LIN {X 0,Y 418.329,Z 253.378,A -85,B 0,C 180,E1 -10089.672,E2 -10089.672} C_VEL
LIN {X 0,Y 418.34,Z 253.367,A -85,B 0,C 180,E1 -10093,E2 -10093} C_VEL
LIN {X 0,Y 418.305,Z 253.377,A -85,B 0,C 180,E1 -10096.734,E2 -10096.734} C_VEL
LIN {X 0,Y 418.264,Z 253.384,A -85,B 0,C 180,E1 -10099.79,E2 -10099.79} C_VEL
LIN {X 0,Y 418.221,Z 253.385,A -85,B 0,C 180,E1 -10102.737,E2 -10102.737} C_VEL
LIN {X 0,Y 418.211,Z 253.382,A -85,B 0,C 180,E1 -10105.908,E2 -10105.908} C_VEL
LIN {X 0,Y 418.25,Z 253.38,A -85,B 0,C 180,E1 -10109.163,E2 -10109.163} C_VEL
LIN {X 0,Y 418.243,Z 253.379,A -85,B 0,C 180,E1 -10112.842,E2 -10112.842} C_VEL
LIN {X 0,Y 418.234,Z 253.386,A -85,B 0,C 180,E1 -10116.237,E2 -10116.237} C_VEL
LIN {X 0,Y 418.194,Z 253.389,A -85,B 0,C 180,E1 -10119.688,E2 -10119.688} C_VEL
LIN {X 0,Y 418.203,Z 253.392,A -85,B 0,C 180,E1 -10122.318,E2 -10122.318} C_VEL
LIN {X 0,Y 418.231,Z 253.389,A -85,B 0,C 180,E1 -10125.109,E2 -10125.109} C_VEL
LIN {X 0,Y 418.214,Z 253.389,A -85,B 0,C 180,E1 -10127.764,E2 -10127.764} C_VEL
LIN {X 0,Y 418.228,Z 253.376,A -85,B 0,C 180,E1 -10131.556,E2 -10131.556} C_VEL
LIN {X 0,Y 418.247,Z 253.374,A -85,B 0,C 180,E1 -10135.158,E2 -10135.158} C_VEL
LIN {X 0,Y 418.237,Z 253.538,A -85,B 0,C 180,E1 -10138.483,E2 -10138.483} C_VEL
LIN {X 0,Y 421.565,Z 267.775,A -85,B 0,C 180,E1 -10141.088,E2 -10141.088} C_VEL
LIN {X 0,Y 422.679,Z 274.559,A -85,B 0,C 180,E1 -10142.254,E2 -10142.254} C_VEL
LIN {X 0,Y 421.513,Z 292.793,A -85,B 0,C 180,E1 -10145.102,E2 -10145.102} C_VEL
LIN {X 0,Y 420.246,Z 314.263,A -85,B 0,C 180,E1 -10148.413,E2 -10148.413} C_VEL
LIN {X 0,Y 419.602,Z 328.237,A -85,B 0,C 180,E1 -10150.523,E2 -10150.523} C_VEL
LIN {X 0,Y 423.082,Z 354.453,A -85,B 0,C 180,E1 -10151.189,E2 -10151.189} C_VEL
LIN {X 0,Y 424.096,Z 367.083,A -85,B 0,C 180,E1 -10151.465,E2 -10151.465} C_VEL
LIN {X 0,Y 423.18,Z 439.314,A -85,B 0,C 180,E1 -10152.731,E2 -10152.731} C_VEL
LIN {X 0,Y 422.504,Z 453.178,A -85,B 0,C 180,E1 -10153.17,E2 -10153.17} C_VEL
LIN {X 0,Y 421.636,Z 466.154,A -85,B 0,C 180,E1 -10153.788,E2 -10153.788} C_VEL
LIN {X 0,Y 420.772,Z 478.778,A -85,B 0,C 180,E1 -10154.624,E2 -10154.624} C_VEL
LIN {X 0,Y 419.851,Z 490.068,A -85,B 0,C 180,E1 -10155.582,E2 -10155.582} C_VEL
LIN {X 0,Y 419.119,Z 500.694,A -85,B 0,C 180,E1 -10156.719,E2 -10156.719} C_VEL
LIN {X 0,Y 418.384,Z 509.542,A -85,B 0,C 180,E1 -10157.879,E2 -10157.879} C_VEL
LIN {X 0,Y 417.84,Z 518.608,A -85,B 0,C 180,E1 -10159.338,E2 -10159.338} C_VEL
LIN {X 0,Y 417.516,Z 525.95,A -85,B 0,C 180,E1 -10160.798,E2 -10160.798} C_VEL
LIN {X 0,Y 417.368,Z 531.851,A -85,B 0,C 180,E1 -10162.258,E2 -10162.258} C_VEL
LIN {X 0,Y 417.325,Z 536.784,A -85,B 0,C 180,E1 -10163.812,E2 -10163.812} C_VEL
LIN {X 0,Y 417.357,Z 540.104,A -85,B 0,C 180,E1 -10165.17,E2 -10165.17} C_VEL
LIN {X 0,Y 417.497,Z 541.913,A -85,B 0,C 180,E1 -10166.139,E2 -10166.139} C_VEL
LIN {X 0,Y 417.534,Z 543.293,A -85,B 0,C 180,E1 -10167.105,E2 -10167.105} C_VEL
LIN {X 0,Y 417.524,Z 544.828,A -85,B 0,C 180,E1 -10169.035,E2 -10169.035} C_VEL
LIN {X 0,Y 417.577,Z 544.955,A -85,B 0,C 180,E1 -10170,E2 -10170} C_VEL
LIN {X 0,Y 417.543,Z 544.671,A -85,B 0,C 180,E1 -10170.964,E2 -10170.964} C_VEL
LIN {X 0,Y 417.521,Z 543.992,A -85,B 0,C 180,E1 -10171.929,E2 -10171.929} C_VEL
LIN {X 0,Y 417.552,Z 542.91,A -85,B 0,C 180,E1 -10172.894,E2 -10172.894} C_VEL
LIN {X 0,Y 417.509,Z 540.432,A -85,B 0,C 180,E1 -10174.344,E2 -10174.344} C_VEL
LIN {X 0,Y 417.444,Z 536.915,A -85,B 0,C 180,E1 -10175.797,E2 -10175.797} C_VEL
LIN {X 0,Y 417.412,Z 532.283,A -85,B 0,C 180,E1 -10177.254,E2 -10177.254} C_VEL
LIN {X 0,Y 417.487,Z 525.258,A -85,B 0,C 180,E1 -10178.958,E2 -10178.958} C_VEL
LIN {X 0,Y 417.764,Z 517.649,A -85,B 0,C 180,E1 -10180.418,E2 -10180.418} C_VEL
LIN {X 0,Y 418.142,Z 509.905,A -85,B 0,C 180,E1 -10181.635,E2 -10181.635} C_VEL
LIN {X 0,Y 418.73,Z 501.162,A -85,B 0,C 180,E1 -10182.774,E2 -10182.774} C_VEL
LIN {X 0,Y 419.276,Z 491.428,A -85,B 0,C 180,E1 -10183.819,E2 -10183.819} C_VEL
LIN {X 0,Y 419.967,Z 480.199,A -85,B 0,C 180,E1 -10184.785,E2 -10184.785} C_VEL
LIN {X 0,Y 420.71,Z 467.631,A -85,B 0,C 180,E1 -10185.626,E2 -10185.626} C_VEL
LIN {X 0,Y 421.417,Z 455.695,A -85,B 0,C 180,E1 -10186.22,E2 -10186.22} C_VEL
LIN {X 0,Y 421.986,Z 442.65,A -85,B 0,C 180,E1 -10186.664,E2 -10186.664} C_VEL
LIN {X 0,Y 422.225,Z 424.048,A -85,B 0,C 180,E1 -10187.028,E2 -10187.028} C_VEL
LIN {X 0,Y 422.691,Z 362.653,A -85,B 0,C 180,E1 -10188.064,E2 -10188.064} C_VEL
LIN {X 0,Y 419.121,Z 329.102,A -85,B 0,C 180,E1 -10188.799,E2 -10188.799} C_VEL
LIN {X 0,Y 419.927,Z 308.584,A -85,B 0,C 180,E1 -10191.862,E2 -10191.862} C_VEL
LIN {X 0,Y 421.052,Z 286.579,A -85,B 0,C 180,E1 -10195.19,E2 -10195.19} C_VEL
LIN {X 0,Y 421.815,Z 271.199,A -85,B 0,C 180,E1 -10197.538,E2 -10197.538} C_VEL
LIN {X 0,Y 418.56,Z 254.958,A -85,B 0,C 180,E1 -10200.246,E2 -10200.246} C_VEL
LIN {X 0,Y 418.271,Z 253.461,A -85,B 0,C 180,E1 -10200.571,E2 -10200.571} C_VEL
LIN {X 0,Y 418.226,Z 253.391,A -85,B 0,C 180,E1 -10203.678,E2 -10203.678} C_VEL
LIN {X 0,Y 418.225,Z 253.39,A -85,B 0,C 180,E1 -10207.224,E2 -10207.224} C_VEL
LIN {X 0,Y 418.199,Z 253.391,A -85,B 0,C 180,E1 -10210.949,E2 -10210.949} C_VEL
LIN {X 0,Y 418.193,Z 253.391,A -85,B 0,C 180,E1 -10213.727,E2 -10213.727} C_VEL
LIN {X 0,Y 418.19,Z 253.39,A -85,B 0,C 180,E1 -10216.446,E2 -10216.446} C_VEL
LIN {X 0,Y 418.198,Z 253.395,A -85,B 0,C 180,E1 -10219.132,E2 -10219.132} C_VEL
LIN {X 0,Y 418.224,Z 253.388,A -85,B 0,C 180,E1 -10222.774,E2 -10222.774} C_VEL
LIN {X 0,Y 418.217,Z 253.386,A -85,B 0,C 180,E1 -10226.32,E2 -10226.32} C_VEL
LIN {X 0,Y 418.226,Z 253.385,A -85,B 0,C 180,E1 -10229.726,E2 -10229.726} C_VEL
LIN {X 0,Y 418.19,Z 253.396,A -85,B 0,C 180,E1 -10233.015,E2 -10233.015} C_VEL
LIN {X 0,Y 418.243,Z 253.383,A -85,B 0,C 180,E1 -10236.216,E2 -10236.216} C_VEL
LIN {X 0,Y 418.235,Z 253.386,A -85,B 0,C 180,E1 -10239.336,E2 -10239.336} C_VEL
LIN {X 0,Y 418.265,Z 253.383,A -85,B 0,C 180,E1 -10242.395,E2 -10242.395} C_VEL
LIN {X 0,Y 418.28,Z 253.379,A -85,B 0,C 180,E1 -10245.402,E2 -10245.402} C_VEL
LIN {X 0,Y 418.298,Z 253.379,A -85,B 0,C 180,E1 -10248.369,E2 -10248.369} C_VEL
LIN {X 0,Y 418.434,Z 253.362,A -85,B 0,C 180,E1 -10252.278,E2 -10252.278} C_VEL
LIN {X 0,Y 418.45,Z 253.36,A -85,B 0,C 180,E1 -10254.217,E2 -10254.217} C_VEL
LIN {X 0,Y 418.523,Z 253.35,A -85,B 0,C 180,E1 -10258.076,E2 -10258.076} C_VEL
LIN {X 0,Y 418.458,Z 253.358,A -85,B 0,C 180,E1 -10260.963,E2 -10260.963} C_VEL
LIN {X 0,Y 418.453,Z 253.359,A -85,B 0,C 180,E1 -10262.888,E2 -10262.888} C_VEL
LIN {X 0,Y 418.424,Z 253.362,A -85,B 0,C 180,E1 -10266.617,E2 -10266.617} C_VEL
LIN {X 0,Y 418.306,Z 253.376,A -85,B 0,C 180,E1 -10269.672,E2 -10269.672} C_VEL
LIN {X 0,Y 418.334,Z 253.372,A -85,B 0,C 180,E1 -10273,E2 -10273} C_VEL
LIN {X 0,Y 418.3,Z 253.377,A -85,B 0,C 180,E1 -10276.735,E2 -10276.735} C_VEL
LIN {X 0,Y 418.259,Z 253.383,A -85,B 0,C 180,E1 -10279.79,E2 -10279.79} C_VEL
LIN {X 0,Y 418.217,Z 253.387,A -85,B 0,C 180,E1 -10282.738,E2 -10282.738} C_VEL
LIN {X 0,Y 418.207,Z 253.392,A -85,B 0,C 180,E1 -10285.909,E2 -10285.909} C_VEL
LIN {X 0,Y 418.247,Z 253.382,A -85,B 0,C 180,E1 -10289.164,E2 -10289.164} C_VEL
LIN {X 0,Y 418.231,Z 253.386,A -85,B 0,C 180,E1 -10292.53,E2 -10292.53} C_VEL
LIN {X 0,Y 418.241,Z 253.383,A -85,B 0,C 180,E1 -10294.843,E2 -10294.843} C_VEL
LIN {X 0,Y 418.224,Z 253.386,A -85,B 0,C 180,E1 -10298.446,E2 -10298.446} C_VEL
LIN {X 0,Y 418.21,Z 253.389,A -85,B 0,C 180,E1 -10302.237,E2 -10302.237} C_VEL
LIN {X 0,Y 418.228,Z 253.385,A -85,B 0,C 180,E1 -10305.11,E2 -10305.11} C_VEL
LIN {X 0,Y 418.212,Z 253.394,A -85,B 0,C 180,E1 -10307.765,E2 -10307.765} C_VEL
LIN {X 0,Y 418.228,Z 253.391,A -85,B 0,C 180,E1 -10311.557,E2 -10311.557} C_VEL
LIN {X 0,Y 418.244,Z 253.385,A -85,B 0,C 180,E1 -10315.159,E2 -10315.159} C_VEL
LIN {X 0,Y 418.229,Z 253.391,A -85,B 0,C 180,E1 -10317.472,E2 -10317.472} C_VEL
LIN {X 0,Y 418.256,Z 253.382,A -85,B 0,C 180,E1 -10320.9,E2 -10320.9} C_VEL
LIN {X 0,Y 418.209,Z 253.388,A -85,B 0,C 180,E1 -10324.093,E2 -10324.093} C_VEL
LIN {X 0,Y 418.232,Z 253.389,A -85,B 0,C 180,E1 -10327.553,E2 -10327.553} C_VEL
LIN {X 0,Y 418.252,Z 253.382,A -85,B 0,C 180,E1 -10330.364,E2 -10330.364} C_VEL
LIN {X 0,Y 418.281,Z 253.384,A -85,B 0,C 180,E1 -10333.404,E2 -10333.404} C_VEL
LIN {X 0,Y 418.349,Z 253.377,A -85,B 0,C 180,E1 -10337.386,E2 -10337.386} C_VEL
LIN {X 0,Y 418.353,Z 253.613,A -85,B 0,C 180,E1 -10339.517,E2 -10339.517} C_VEL
LIN {X 0,Y 418.633,Z 254.814,A -85,B 0,C 180,E1 -10339.664,E2 -10339.664} C_VEL
LIN {X 0,Y 423.488,Z 268.312,A -85,B 0,C 180,E1 -10340.107,E2 -10340.107} C_VEL
LIN {X 0,Y 422.736,Z 341.816,A -85,B 0,C 180,E1 -10341.375,E2 -10341.375} C_VEL
LIN {X 0,Y 422.651,Z 355.208,A -85,B 0,C 180,E1 -10341.815,E2 -10341.815} C_VEL
LIN {X 0,Y 422.338,Z 366.469,A -85,B 0,C 180,E1 -10342.35,E2 -10342.35} C_VEL
LIN {X 0,Y 421.96,Z 377.78,A -85,B 0,C 180,E1 -10343.065,E2 -10343.065} C_VEL
LIN {X 0,Y 421.365,Z 389.414,A -85,B 0,C 180,E1 -10344.017,E2 -10344.017} C_VEL
LIN {X 0,Y 420.76,Z 399.809,A -85,B 0,C 180,E1 -10345.09,E2 -10345.09} C_VEL
LIN {X 0,Y 420.249,Z 408.305,A -85,B 0,C 180,E1 -10346.165,E2 -10346.165} C_VEL
LIN {X 0,Y 419.828,Z 414.206,A -85,B 0,C 180,E1 -10347.043,E2 -10347.043} C_VEL
LIN {X 0,Y 418.927,Z 418,A -85,B 0,C 180,E1 -10347.654,E2 -10347.654} C_VEL
LIN {X 0,Y 415.715,Z 423.87,A -85,B 0,C 180,E1 -10348.66,E2 -10348.66} C_VEL
LIN {X 0,Y 412.503,Z 429.122,A -85,B 0,C 180,E1 -10349.735,E2 -10349.735} C_VEL
LIN {X 0,Y 411.616,Z 431.916,A -85,B 0,C 180,E1 -10350.444,E2 -10350.444} C_VEL
LIN {X 0,Y 411.325,Z 436.709,A -85,B 0,C 180,E1 -10351.959,E2 -10351.959} C_VEL
LIN {X 0,Y 411.028,Z 440.273,A -85,B 0,C 180,E1 -10353.431,E2 -10353.431} C_VEL
LIN {X 0,Y 411.014,Z 442.819,A -85,B 0,C 180,E1 -10354.905,E2 -10354.905} C_VEL
LIN {X 0,Y 410.93,Z 444.038,A -85,B 0,C 180,E1 -10355.89,E2 -10355.89} C_VEL
LIN {X 0,Y 410.866,Z 444.998,A -85,B 0,C 180,E1 -10357.198,E2 -10357.198} C_VEL
LIN {X 0,Y 410.864,Z 445.251,A -85,B 0,C 180,E1 -10358.856,E2 -10358.856} C_VEL
LIN {X 0,Y 410.918,Z 444.89,A -85,B 0,C 180,E1 -10359.848,E2 -10359.848} C_VEL
LIN {X 0,Y 410.983,Z 444.108,A -85,B 0,C 180,E1 -10360.842,E2 -10360.842} C_VEL
LIN {X 0,Y 411.326,Z 441.302,A -85,B 0,C 180,E1 -10362.834,E2 -10362.834} C_VEL
LIN {X 0,Y 411.645,Z 438.051,A -85,B 0,C 180,E1 -10364.333,E2 -10364.333} C_VEL
LIN {X 0,Y 412.072,Z 433.706,A -85,B 0,C 180,E1 -10365.836,E2 -10365.836} C_VEL
LIN {X 0,Y 412.7,Z 427.4,A -85,B 0,C 180,E1 -10367.512,E2 -10367.512} C_VEL
LIN {X 0,Y 413.481,Z 419.712,A -85,B 0,C 180,E1 -10369.099,E2 -10369.099} C_VEL
LIN {X 0,Y 414.137,Z 412.184,A -85,B 0,C 180,E1 -10370.358,E2 -10370.358} C_VEL
LIN {X 0,Y 414.964,Z 402.642,A -85,B 0,C 180,E1 -10371.659,E2 -10371.659} C_VEL
LIN {X 0,Y 415.666,Z 392.66,A -85,B 0,C 180,E1 -10372.753,E2 -10372.753} C_VEL
LIN {X 0,Y 416.294,Z 382.696,A -85,B 0,C 180,E1 -10373.638,E2 -10373.638} C_VEL
LIN {X 0,Y 416.958,Z 370.814,A -85,B 0,C 180,E1 -10374.467,E2 -10374.467} C_VEL
LIN {X 0,Y 417.371,Z 358.128,A -85,B 0,C 180,E1 -10375.128,E2 -10375.128} C_VEL
LIN {X 0,Y 417.56,Z 345.349,A -85,B 0,C 180,E1 -10375.583,E2 -10375.583} C_VEL
LIN {X 0,Y 417.672,Z 324.353,A -85,B 0,C 180,E1 -10376.004,E2 -10376.004} C_VEL
LIN {X 0,Y 418.487,Z 271.987,A -85,B 0,C 180,E1 -10376.91,E2 -10376.91} C_VEL
LIN {X 0,Y 411.384,Z 255.243,A -85,B 0,C 180,E1 -10377.651,E2 -10377.651} C_VEL
LIN {X 0,Y 411.205,Z 254.336,A -85,B 0,C 180,E1 -10377.862,E2 -10377.862} C_VEL
LIN {X 0,Y 411.19,Z 254.242,A -85,B 0,C 180,E1 -10380.847,E2 -10380.847} C_VEL
LIN {X 0,Y 411.194,Z 254.26,A -85,B 0,C 180,E1 -10384.334,E2 -10384.334} C_VEL
LIN {X 0,Y 411.188,Z 254.232,A -85,B 0,C 180,E1 -10386.742,E2 -10386.742} C_VEL
LIN {X 0,Y 411.168,Z 254.268,A -85,B 0,C 180,E1 -10389.719,E2 -10389.719} C_VEL
LIN {X 0,Y 411.162,Z 254.269,A -85,B 0,C 180,E1 -10393.134,E2 -10393.134} C_VEL
LIN {X 0,Y 411.162,Z 254.263,A -85,B 0,C 180,E1 -10395.881,E2 -10395.881} C_VEL
LIN {X 0,Y 411.146,Z 254.273,A -85,B 0,C 180,E1 -10398.774,E2 -10398.774} C_VEL
LIN {X 0,Y 411.179,Z 254.251,A -85,B 0,C 180,E1 -10402.024,E2 -10402.024} C_VEL
LIN {X 0,Y 411.202,Z 254.263,A -85,B 0,C 180,E1 -10405.666,E2 -10405.666} C_VEL
LIN {X 0,Y 411.185,Z 254.243,A -85,B 0,C 180,E1 -10409.152,E2 -10409.152} C_VEL
LIN {X 0,Y 411.172,Z 254.257,A -85,B 0,C 180,E1 -10411.406,E2 -10411.406} C_VEL
LIN {X 0,Y 411.212,Z 254.258,A -85,B 0,C 180,E1 -10414.932,E2 -10414.932} C_VEL
LIN {X 0,Y 411.199,Z 254.235,A -85,B 0,C 180,E1 -10417.913,E2 -10417.913} C_VEL
LIN {X 0,Y 411.217,Z 254.254,A -85,B 0,C 180,E1 -10421.051,E2 -10421.051} C_VEL
LIN {X 0,Y 411.247,Z 254.255,A -85,B 0,C 180,E1 -10424.131,E2 -10424.131} C_VEL
LIN {X 0,Y 411.297,Z 254.248,A -85,B 0,C 180,E1 -10427.165,E2 -10427.165} C_VEL
LIN {X 0,Y 411.281,Z 254.245,A -85,B 0,C 180,E1 -10430.161,E2 -10430.161} C_VEL
LIN {X 0,Y 411.383,Z 254.239,A -85,B 0,C 180,E1 -10433.131,E2 -10433.131} C_VEL
LIN {X 0,Y 411.278,Z 254.25,A -85,B 0,C 180,E1 -10435.098,E2 -10435.098} C_VEL
LIN {X 0,Y 411.494,Z 254.228,A -85,B 0,C 180,E1 -10438.042,E2 -10438.042} C_VEL
LIN {X 0,Y 411.369,Z 254.237,A -85,B 0,C 180,E1 -10440.979,E2 -10440.979} C_VEL
LIN {X 0,Y 411.431,Z 254.227,A -85,B 0,C 180,E1 -10442.937,E2 -10442.937} C_VEL
LIN {X 0,Y 411.378,Z 254.235,A -85,B 0,C 180,E1 -10446.868,E2 -10446.868} C_VEL
LIN {X 0,Y 411.281,Z 254.254,A -85,B 0,C 180,E1 -10449.839,E2 -10449.839} C_VEL
LIN {X 0,Y 411.299,Z 254.244,A -85,B 0,C 180,E1 -10453.104,E2 -10453.104} C_VEL
LIN {X 0,Y 411.252,Z 254.257,A -85,B 0,C 180,E1 -10456.889,E2 -10456.889} C_VEL
LIN {X 0,Y 411.225,Z 254.259,A -85,B 0,C 180,E1 -10459.987,E2 -10459.987} C_VEL
LIN {X 0,Y 411.181,Z 254.266,A -85,B 0,C 180,E1 -10463.149,E2 -10463.149} C_VEL
LIN {X 0,Y 411.165,Z 254.26,A -85,B 0,C 180,E1 -10466.386,E2 -10466.386} C_VEL
LIN {X 0,Y 411.189,Z 254.264,A -85,B 0,C 180,E1 -10469.714,E2 -10469.714} C_VEL
LIN {X 0,Y 411.199,Z 254.253,A -85,B 0,C 180,E1 -10473.156,E2 -10473.156} C_VEL
LIN {X 0,Y 411.184,Z 254.267,A -85,B 0,C 180,E1 -10476.552,E2 -10476.552} C_VEL
LIN {X 0,Y 411.163,Z 254.265,A -85,B 0,C 180,E1 -10479.72,E2 -10479.72} C_VEL
LIN {X 0,Y 411.158,Z 254.264,A -85,B 0,C 180,E1 -10483.136,E2 -10483.136} C_VEL
LIN {X 0,Y 411.159,Z 254.266,A -85,B 0,C 180,E1 -10485.882,E2 -10485.882} C_VEL
LIN {X 0,Y 411.154,Z 254.262,A -85,B 0,C 180,E1 -10489.493,E2 -10489.493} C_VEL
LIN {X 0,Y 411.176,Z 254.261,A -85,B 0,C 180,E1 -10492.025,E2 -10492.025} C_VEL
LIN {X 0,Y 411.199,Z 254.252,A -85,B 0,C 180,E1 -10495.124,E2 -10495.124} C_VEL
LIN {X 0,Y 411.228,Z 254.442,A -85,B 0,C 180,E1 -10498.148,E2 -10498.148} C_VEL
LIN {X 0,Y 414.174,Z 267.128,A -85,B 0,C 180,E1 -10500.522,E2 -10500.522} C_VEL
LIN {X 0,Y 415.815,Z 275.627,A -85,B 0,C 180,E1 -10502.029,E2 -10502.029} C_VEL
LIN {X 0,Y 414.635,Z 293.851,A -85,B 0,C 180,E1 -10504.929,E2 -10504.929} C_VEL
LIN {X 0,Y 413.205,Z 316.945,A -85,B 0,C 180,E1 -10508.55,E2 -10508.55} C_VEL
LIN {X 0,Y 412.71,Z 327.289,A -85,B 0,C 180,E1 -10510.132,E2 -10510.132} C_VEL
LIN {X 0,Y 416.221,Z 353.382,A -85,B 0,C 180,E1 -10510.821,E2 -10510.821} C_VEL
LIN {X 0,Y 417.433,Z 366.101,A -85,B 0,C 180,E1 -10511.114,E2 -10511.114} C_VEL
LIN {X 0,Y 416.44,Z 438.793,A -85,B 0,C 180,E1 -10512.411,E2 -10512.411} C_VEL
LIN {X 0,Y 415.764,Z 452.537,A -85,B 0,C 180,E1 -10512.857,E2 -10512.857} C_VEL
LIN {X 0,Y 414.898,Z 464.922,A -85,B 0,C 180,E1 -10513.454,E2 -10513.454} C_VEL
LIN {X 0,Y 414.034,Z 476.832,A -85,B 0,C 180,E1 -10514.241,E2 -10514.241} C_VEL
LIN {X 0,Y 413.079,Z 488.314,A -85,B 0,C 180,E1 -10515.214,E2 -10515.214} C_VEL
LIN {X 0,Y 412.292,Z 497.634,A -85,B 0,C 180,E1 -10516.193,E2 -10516.193} C_VEL
LIN {X 0,Y 411.597,Z 507.261,A -85,B 0,C 180,E1 -10517.426,E2 -10517.426} C_VEL
LIN {X 0,Y 410.939,Z 516.573,A -85,B 0,C 180,E1 -10518.907,E2 -10518.907} C_VEL
LIN {X 0,Y 410.492,Z 524.111,A -85,B 0,C 180,E1 -10520.391,E2 -10520.391} C_VEL
LIN {X 0,Y 410.29,Z 531.109,A -85,B 0,C 180,E1 -10522.123,E2 -10522.123} C_VEL
LIN {X 0,Y 410.314,Z 535.287,A -85,B 0,C 180,E1 -10523.437,E2 -10523.437} C_VEL
LIN {X 0,Y 410.279,Z 539.315,A -85,B 0,C 180,E1 -10525.086,E2 -10525.086} C_VEL
LIN {X 0,Y 410.427,Z 541.11,A -85,B 0,C 180,E1 -10526.072,E2 -10526.072} C_VEL
LIN {X 0,Y 410.483,Z 542.481,A -85,B 0,C 180,E1 -10527.055,E2 -10527.055} C_VEL
LIN {X 0,Y 410.436,Z 543.437,A -85,B 0,C 180,E1 -10528.037,E2 -10528.037} C_VEL
LIN {X 0,Y 410.471,Z 543.986,A -85,B 0,C 180,E1 -10529.019,E2 -10529.019} C_VEL
LIN {X 0,Y 410.528,Z 544.099,A -85,B 0,C 180,E1 -10530,E2 -10530} C_VEL
LIN {X 0,Y 410.492,Z 543.805,A -85,B 0,C 180,E1 -10530.981,E2 -10530.981} C_VEL
LIN {X 0,Y 410.47,Z 543.114,A -85,B 0,C 180,E1 -10531.962,E2 -10531.962} C_VEL
LIN {X 0,Y 410.503,Z 542.012,A -85,B 0,C 180,E1 -10532.944,E2 -10532.944} C_VEL
LIN {X 0,Y 410.443,Z 539.513,A -85,B 0,C 180,E1 -10534.419,E2 -10534.419} C_VEL
LIN {X 0,Y 410.378,Z 534.748,A -85,B 0,C 180,E1 -10536.316,E2 -10536.316} C_VEL
LIN {X 0,Y 410.333,Z 529.453,A -85,B 0,C 180,E1 -10537.875,E2 -10537.875} C_VEL
LIN {X 0,Y 410.494,Z 523.089,A -85,B 0,C 180,E1 -10539.36,E2 -10539.36} C_VEL
LIN {X 0,Y 410.813,Z 515.154,A -85,B 0,C 180,E1 -10540.846,E2 -10540.846} C_VEL
LIN {X 0,Y 411.373,Z 505.235,A -85,B 0,C 180,E1 -10542.33,E2 -10542.33} C_VEL
LIN {X 0,Y 411.908,Z 495.947,A -85,B 0,C 180,E1 -10543.458,E2 -10543.458} C_VEL
LIN {X 0,Y 412.624,Z 484.831,A -85,B 0,C 180,E1 -10544.549,E2 -10544.549} C_VEL
LIN {X 0,Y 413.411,Z 473.825,A -85,B 0,C 180,E1 -10545.403,E2 -10545.403} C_VEL
LIN {X 0,Y 414.149,Z 461.68,A -85,B 0,C 180,E1 -10546.133,E2 -10546.133} C_VEL
LIN {X 0,Y 414.796,Z 449.272,A -85,B 0,C 180,E1 -10546.676,E2 -10546.676} C_VEL
LIN {X 0,Y 415.238,Z 436.492,A -85,B 0,C 180,E1 -10547.038,E2 -10547.038} C_VEL
LIN {X 0,Y 415.864,Z 363.556,A -85,B 0,C 180,E1 -10548.301,E2 -10548.301} C_VEL
LIN {X 0,Y 412.124,Z 328.112,A -85,B 0,C 180,E1 -10549.098,E2 -10549.098} C_VEL
LIN {X 0,Y 413,Z 307.432,A -85,B 0,C 180,E1 -10552.248,E2 -10552.248} C_VEL
LIN {X 0,Y 414.179,Z 285.781,A -85,B 0,C 180,E1 -10555.579,E2 -10555.579} C_VEL
LIN {X 0,Y 414.84,Z 273.589,A -85,B 0,C 180,E1 -10557.469,E2 -10557.469} C_VEL
LIN {X 0,Y 413.688,Z 266.297,A -85,B 0,C 180,E1 -10558.68,E2 -10558.68} C_VEL
LIN {X 0,Y 411.244,Z 254.369,A -85,B 0,C 180,E1 -10560.77,E2 -10560.77} C_VEL
LIN {X 0,Y 411.186,Z 254.266,A -85,B 0,C 180,E1 -10564.334,E2 -10564.334} C_VEL
LIN {X 0,Y 411.179,Z 254.264,A -85,B 0,C 180,E1 -10566.742,E2 -10566.742} C_VEL
LIN {X 0,Y 411.156,Z 254.268,A -85,B 0,C 180,E1 -10569.718,E2 -10569.718} C_VEL
LIN {X 0,Y 411.153,Z 254.271,A -85,B 0,C 180,E1 -10573.134,E2 -10573.134} C_VEL
LIN {X 0,Y 411.155,Z 254.267,A -85,B 0,C 180,E1 -10575.881,E2 -10575.881} C_VEL
LIN {X 0,Y 411.149,Z 254.27,A -85,B 0,C 180,E1 -10579.492,E2 -10579.492} C_VEL
LIN {X 0,Y 411.173,Z 254.264,A -85,B 0,C 180,E1 -10582.024,E2 -10582.024} C_VEL
LIN {X 0,Y 411.19,Z 254.268,A -85,B 0,C 180,E1 -10585.123,E2 -10585.123} C_VEL
LIN {X 0,Y 411.143,Z 254.267,A -85,B 0,C 180,E1 -10588.001,E2 -10588.001} C_VEL
LIN {X 0,Y 411.158,Z 254.268,A -85,B 0,C 180,E1 -10591.405,E2 -10591.405} C_VEL
LIN {X 0,Y 411.176,Z 254.27,A -85,B 0,C 180,E1 -10594.941,E2 -10594.941} C_VEL
LIN {X 0,Y 411.19,Z 254.261,A -85,B 0,C 180,E1 -10597.913,E2 -10597.913} C_VEL
LIN {X 0,Y 411.205,Z 254.264,A -85,B 0,C 180,E1 -10601.051,E2 -10601.051} C_VEL
LIN {X 0,Y 411.233,Z 254.257,A -85,B 0,C 180,E1 -10604.131,E2 -10604.131} C_VEL
LIN {X 0,Y 411.291,Z 254.251,A -85,B 0,C 180,E1 -10607.165,E2 -10607.165} C_VEL
LIN {X 0,Y 411.267,Z 254.253,A -85,B 0,C 180,E1 -10610.161,E2 -10610.161} C_VEL
LIN {X 0,Y 411.372,Z 254.24,A -85,B 0,C 180,E1 -10613.132,E2 -10613.132} C_VEL
LIN {X 0,Y 411.272,Z 254.253,A -85,B 0,C 180,E1 -10615.099,E2 -10615.099} C_VEL
LIN {X 0,Y 411.492,Z 254.226,A -85,B 0,C 180,E1 -10618.043,E2 -10618.043} C_VEL
LIN {X 0,Y 411.487,Z 254.226,A -85,B 0,C 180,E1 -10621.958,E2 -10621.958} C_VEL
LIN {X 0,Y 411.372,Z 254.239,A -85,B 0,C 180,E1 -10626.618,E2 -10626.618} C_VEL
LIN {X 0,Y 411.293,Z 254.25,A -85,B 0,C 180,E1 -10628.847,E2 -10628.847} C_VEL
LIN {X 0,Y 411.26,Z 254.255,A -85,B 0,C 180,E1 -10631.834,E2 -10631.834} C_VEL
LIN {X 0,Y 411.241,Z 254.256,A -85,B 0,C 180,E1 -10634.854,E2 -10634.854} C_VEL
LIN {X 0,Y 411.233,Z 254.26,A -85,B 0,C 180,E1 -10637.916,E2 -10637.916} C_VEL
LIN {X 0,Y 411.185,Z 254.262,A -85,B 0,C 180,E1 -10641.035,E2 -10641.035} C_VEL
LIN {X 0,Y 411.18,Z 254.268,A -85,B 0,C 180,E1 -10644.219,E2 -10644.219} C_VEL
LIN {X 0,Y 411.136,Z 254.269,A -85,B 0,C 180,E1 -10647.487,E2 -10647.487} C_VEL
LIN {X 0,Y 411.186,Z 254.265,A -85,B 0,C 180,E1 -10649.714,E2 -10649.714} C_VEL
LIN {X 0,Y 411.196,Z 254.261,A -85,B 0,C 180,E1 -10653.157,E2 -10653.157} C_VEL
LIN {X 0,Y 411.18,Z 254.263,A -85,B 0,C 180,E1 -10656.553,E2 -10656.553} C_VEL
LIN {X 0,Y 411.159,Z 254.271,A -85,B 0,C 180,E1 -10659.721,E2 -10659.721} C_VEL
LIN {X 0,Y 411.155,Z 254.266,A -85,B 0,C 180,E1 -10663.137,E2 -10663.137} C_VEL
LIN {X 0,Y 411.157,Z 254.271,A -85,B 0,C 180,E1 -10665.883,E2 -10665.883} C_VEL
LIN {X 0,Y 411.152,Z 254.271,A -85,B 0,C 180,E1 -10669.494,E2 -10669.494} C_VEL
LIN {X 0,Y 411.176,Z 254.266,A -85,B 0,C 180,E1 -10672.026,E2 -10672.026} C_VEL
LIN {X 0,Y 411.196,Z 254.263,A -85,B 0,C 180,E1 -10675.125,E2 -10675.125} C_VEL
LIN {X 0,Y 411.151,Z 254.268,A -85,B 0,C 180,E1 -10678.003,E2 -10678.003} C_VEL
LIN {X 0,Y 411.167,Z 254.27,A -85,B 0,C 180,E1 -10681.407,E2 -10681.407} C_VEL
LIN {X 0,Y 411.187,Z 254.264,A -85,B 0,C 180,E1 -10684.943,E2 -10684.943} C_VEL
LIN {X 0,Y 411.2,Z 254.262,A -85,B 0,C 180,E1 -10687.914,E2 -10687.914} C_VEL
LIN {X 0,Y 411.19,Z 254.265,A -85,B 0,C 180,E1 -10691.051,E2 -10691.051} C_VEL
LIN {X 0,Y 411.199,Z 254.26,A -85,B 0,C 180,E1 -10694.13,E2 -10694.13} C_VEL
LIN {X 0,Y 411.298,Z 254.252,A -85,B 0,C 180,E1 -10697.166,E2 -10697.166} C_VEL
LIN {X 0,Y 411.305,Z 254.438,A -85,B 0,C 180,E1 -10699.216,E2 -10699.216} C_VEL
LIN {X 0,Y 411.451,Z 255.25,A -85,B 0,C 180,E1 -10699.359,E2 -10699.359} C_VEL
LIN {X 0,Y 416.769,Z 270.131,A -85,B 0,C 180,E1 -10699.865,E2 -10699.865} C_VEL
LIN {X 0,Y 415.912,Z 341.892,A -85,B 0,C 180,E1 -10701.113,E2 -10701.113} C_VEL
LIN {X 0,Y 415.833,Z 354.716,A -85,B 0,C 180,E1 -10701.527,E2 -10701.527} C_VEL
LIN {X 0,Y 415.49,Z 366.877,A -85,B 0,C 180,E1 -10702.101,E2 -10702.101} C_VEL
LIN {X 0,Y 415.102,Z 378.281,A -85,B 0,C 180,E1 -10702.828,E2 -10702.828} C_VEL
LIN {X 0,Y 414.481,Z 390.009,A -85,B 0,C 180,E1 -10703.795,E2 -10703.795} C_VEL
LIN {X 0,Y 413.848,Z 400.449,A -85,B 0,C 180,E1 -10704.885,E2 -10704.885} C_VEL
LIN {X 0,Y 413.272,Z 409.85,A -85,B 0,C 180,E1 -10706.1,E2 -10706.1} C_VEL
LIN {X 0,Y 412.706,Z 417.574,A -85,B 0,C 180,E1 -10707.316,E2 -10707.316} C_VEL
LIN {X 0,Y 412.092,Z 425.134,A -85,B 0,C 180,E1 -10708.779,E2 -10708.779} C_VEL
LIN {X 0,Y 411.616,Z 431.916,A -85,B 0,C 180,E1 -10710.444,E2 -10710.444} C_VEL
LIN {X 0,Y 410.74,Z 434.523,A -85,B 0,C 180,E1 -10711.174,E2 -10711.174} C_VEL
LIN {X 0,Y 406.248,Z 439.724,A -85,B 0,C 180,E1 -10712.87,E2 -10712.87} C_VEL
LIN {X 0,Y 404.233,Z 442.061,A -85,B 0,C 180,E1 -10713.903,E2 -10713.903} C_VEL
LIN {X 0,Y 403.925,Z 442.96,A -85,B 0,C 180,E1 -10714.444,E2 -10714.444} C_VEL
LIN {X 0,Y 403.876,Z 444.991,A -85,B 0,C 180,E1 -10715.993,E2 -10715.993} C_VEL
LIN {X 0,Y 403.799,Z 446.102,A -85,B 0,C 180,E1 -10718.004,E2 -10718.004} C_VEL
LIN {X 0,Y 403.848,Z 446.086,A -85,B 0,C 180,E1 -10719.011,E2 -10719.011} C_VEL
LIN {X 0,Y 403.897,Z 445.686,A -85,B 0,C 180,E1 -10720.021,E2 -10720.021} C_VEL
LIN {X 0,Y 404.135,Z 443.617,A -85,B 0,C 180,E1 -10722.045,E2 -10722.045} C_VEL
LIN {X 0,Y 404.403,Z 441.54,A -85,B 0,C 180,E1 -10723.29,E2 -10723.29} C_VEL
LIN {X 0,Y 404.823,Z 437.301,A -85,B 0,C 180,E1 -10725.094,E2 -10725.094} C_VEL
LIN {X 0,Y 405.353,Z 432.476,A -85,B 0,C 180,E1 -10726.623,E2 -10726.623} C_VEL
LIN {X 0,Y 405.982,Z 426.348,A -85,B 0,C 180,E1 -10728.156,E2 -10728.156} C_VEL
LIN {X 0,Y 406.807,Z 418.626,A -85,B 0,C 180,E1 -10729.687,E2 -10729.687} C_VEL
LIN {X 0,Y 407.571,Z 410.658,A -85,B 0,C 180,E1 -10730.965,E2 -10730.965} C_VEL
LIN {X 0,Y 408.378,Z 400.862,A -85,B 0,C 180,E1 -10732.248,E2 -10732.248} C_VEL
LIN {X 0,Y 409.154,Z 391.185,A -85,B 0,C 180,E1 -10733.27,E2 -10733.27} C_VEL
LIN {X 0,Y 409.84,Z 380.682,A -85,B 0,C 180,E1 -10734.168,E2 -10734.168} C_VEL
LIN {X 0,Y 410.457,Z 368.828,A -85,B 0,C 180,E1 -10734.952,E2 -10734.952} C_VEL
LIN {X 0,Y 410.829,Z 356.149,A -85,B 0,C 180,E1 -10735.574,E2 -10735.574} C_VEL
LIN {X 0,Y 410.973,Z 343.681,A -85,B 0,C 180,E1 -10735.99,E2 -10735.99} C_VEL
LIN {X 0,Y 411.355,Z 306.087,A -85,B 0,C 180,E1 -10736.684,E2 -10736.684} C_VEL
LIN {X 0,Y 411.883,Z 273.341,A -85,B 0,C 180,E1 -10737.261,E2 -10737.261} C_VEL
LIN {X 0,Y 404.311,Z 256.008,A -85,B 0,C 180,E1 -10738.068,E2 -10738.068} C_VEL
LIN {X 0,Y 404.173,Z 255.199,A -85,B 0,C 180,E1 -10738.283,E2 -10738.283} C_VEL
LIN {X 0,Y 404.14,Z 255.12,A -85,B 0,C 180,E1 -10741.557,E2 -10741.557} C_VEL
LIN {X 0,Y 404.174,Z 255.12,A -85,B 0,C 180,E1 -10745.017,E2 -10745.017} C_VEL
LIN {X 0,Y 404.134,Z 255.136,A -85,B 0,C 180,E1 -10748.759,E2 -10748.759} C_VEL
LIN {X 0,Y 404.106,Z 255.139,A -85,B 0,C 180,E1 -10751.596,E2 -10751.596} C_VEL
LIN {X 0,Y 404.142,Z 255.147,A -85,B 0,C 180,E1 -10754.521,E2 -10754.521} C_VEL
LIN {X 0,Y 404.119,Z 255.134,A -85,B 0,C 180,E1 -10757.293,E2 -10757.293} C_VEL
LIN {X 0,Y 404.131,Z 255.145,A -85,B 0,C 180,E1 -10759.95,E2 -10759.95} C_VEL
LIN {X 0,Y 404.128,Z 255.13,A -85,B 0,C 180,E1 -10763.126,E2 -10763.126} C_VEL
LIN {X 0,Y 404.142,Z 255.148,A -85,B 0,C 180,E1 -10766.187,E2 -10766.187} C_VEL
LIN {X 0,Y 404.14,Z 255.118,A -85,B 0,C 180,E1 -10769.714,E2 -10769.714} C_VEL
LIN {X 0,Y 404.115,Z 255.145,A -85,B 0,C 180,E1 -10773.117,E2 -10773.117} C_VEL
LIN {X 0,Y 404.152,Z 255.124,A -85,B 0,C 180,E1 -10776.424,E2 -10776.424} C_VEL
LIN {X 0,Y 404.187,Z 255.117,A -85,B 0,C 180,E1 -10779.874,E2 -10779.874} C_VEL
LIN {X 0,Y 404.211,Z 255.132,A -85,B 0,C 180,E1 -10782.993,E2 -10782.993} C_VEL
LIN {X 0,Y 404.278,Z 255.122,A -85,B 0,C 180,E1 -10786.938,E2 -10786.938} C_VEL
LIN {X 0,Y 404.247,Z 255.122,A -85,B 0,C 180,E1 -10789.988,E2 -10789.988} C_VEL
LIN {X 0,Y 404.334,Z 255.116,A -85,B 0,C 180,E1 -10793.011,E2 -10793.011} C_VEL
LIN {X 0,Y 404.249,Z 255.125,A -85,B 0,C 180,E1 -10795.013,E2 -10795.013} C_VEL
LIN {X 0,Y 404.463,Z 255.104,A -85,B 0,C 180,E1 -10798.008,E2 -10798.008} C_VEL
LIN {X 0,Y 404.34,Z 255.113,A -85,B 0,C 180,E1 -10800.996,E2 -10800.996} C_VEL
LIN {X 0,Y 404.39,Z 255.104,A -85,B 0,C 180,E1 -10802.988,E2 -10802.988} C_VEL
LIN {X 0,Y 404.329,Z 255.114,A -85,B 0,C 180,E1 -10806.988,E2 -10806.988} C_VEL
LIN {X 0,Y 404.247,Z 255.129,A -85,B 0,C 180,E1 -10810.012,E2 -10810.012} C_VEL
LIN {X 0,Y 404.261,Z 255.12,A -85,B 0,C 180,E1 -10813.211,E2 -10813.211} C_VEL
LIN {X 0,Y 404.21,Z 255.135,A -85,B 0,C 180,E1 -10817.007,E2 -10817.007} C_VEL
LIN {X 0,Y 404.158,Z 255.139,A -85,B 0,C 180,E1 -10820.352,E2 -10820.352} C_VEL
LIN {X 0,Y 404.142,Z 255.145,A -85,B 0,C 180,E1 -10823.576,E2 -10823.576} C_VEL
LIN {X 0,Y 404.097,Z 255.135,A -85,B 0,C 180,E1 -10826.884,E2 -10826.884} C_VEL
LIN {X 0,Y 404.136,Z 255.142,A -85,B 0,C 180,E1 -10830.286,E2 -10830.286} C_VEL
LIN {X 0,Y 404.133,Z 255.13,A -85,B 0,C 180,E1 -10833.813,E2 -10833.813} C_VEL
LIN {X 0,Y 404.127,Z 255.148,A -85,B 0,C 180,E1 -10836.874,E2 -10836.874} C_VEL
LIN {X 0,Y 404.113,Z 255.143,A -85,B 0,C 180,E1 -10840.075,E2 -10840.075} C_VEL
LIN {X 0,Y 404.137,Z 255.138,A -85,B 0,C 180,E1 -10843.082,E2 -10843.082} C_VEL
LIN {X 0,Y 404.116,Z 255.144,A -85,B 0,C 180,E1 -10845.922,E2 -10845.922} C_VEL
LIN {X 0,Y 404.098,Z 255.149,A -85,B 0,C 180,E1 -10848.633,E2 -10848.633} C_VEL
LIN {X 0,Y 404.133,Z 255.129,A -85,B 0,C 180,E1 -10851.496,E2 -10851.496} C_VEL
LIN {X 0,Y 404.17,Z 255.126,A -85,B 0,C 180,E1 -10854.983,E2 -10854.983} C_VEL
LIN {X 0,Y 404.184,Z 255.314,A -85,B 0,C 180,E1 -10857.784,E2 -10857.784} C_VEL
LIN {X 0,Y 407.221,Z 268.196,A -85,B 0,C 180,E1 -10860.253,E2 -10860.253} C_VEL
LIN {X 0,Y 408.946,Z 276.837,A -85,B 0,C 180,E1 -10861.82,E2 -10861.82} C_VEL
LIN {X 0,Y 407.749,Z 294.911,A -85,B 0,C 180,E1 -10864.749,E2 -10864.749} C_VEL
LIN {X 0,Y 406.247,Z 317.983,A -85,B 0,C 180,E1 -10868.431,E2 -10868.431} C_VEL
LIN {X 0,Y 405.818,Z 326.452,A -85,B 0,C 180,E1 -10869.735,E2 -10869.735} C_VEL
LIN {X 0,Y 409.518,Z 353.514,A -85,B 0,C 180,E1 -10870.471,E2 -10870.471} C_VEL
LIN {X 0,Y 410.785,Z 366.656,A -85,B 0,C 180,E1 -10870.781,E2 -10870.781} C_VEL
LIN {X 0,Y 409.785,Z 437.186,A -85,B 0,C 180,E1 -10872.051,E2 -10872.051} C_VEL
LIN {X 0,Y 409.194,Z 450.411,A -85,B 0,C 180,E1 -10872.476,E2 -10872.476} C_VEL
LIN {X 0,Y 408.236,Z 463.704,A -85,B 0,C 180,E1 -10873.111,E2 -10873.111} C_VEL
LIN {X 0,Y 407.335,Z 474.906,A -85,B 0,C 180,E1 -10873.846,E2 -10873.846} C_VEL
LIN {X 0,Y 406.289,Z 486.573,A -85,B 0,C 180,E1 -10874.833,E2 -10874.833} C_VEL
LIN {X 0,Y 405.366,Z 497.118,A -85,B 0,C 180,E1 -10875.953,E2 -10875.953} C_VEL
LIN {X 0,Y 404.65,Z 506.675,A -85,B 0,C 180,E1 -10877.206,E2 -10877.206} C_VEL
LIN {X 0,Y 403.919,Z 515.923,A -85,B 0,C 180,E1 -10878.712,E2 -10878.712} C_VEL
LIN {X 0,Y 403.434,Z 523.422,A -85,B 0,C 180,E1 -10880.221,E2 -10880.221} C_VEL
LIN {X 0,Y 403.209,Z 530.37,A -85,B 0,C 180,E1 -10881.984,E2 -10881.984} C_VEL
LIN {X 0,Y 403.236,Z 534.861,A -85,B 0,C 180,E1 -10883.441,E2 -10883.441} C_VEL
LIN {X 0,Y 403.206,Z 538.527,A -85,B 0,C 180,E1 -10885,E2 -10885} C_VEL
LIN {X 0,Y 403.358,Z 540.309,A -85,B 0,C 180,E1 -10886.003,E2 -10886.003} C_VEL
LIN {X 0,Y 403.432,Z 541.671,A -85,B 0,C 180,E1 -10887.004,E2 -10887.004} C_VEL
LIN {X 0,Y 403.38,Z 542.616,A -85,B 0,C 180,E1 -10888.003,E2 -10888.003} C_VEL
LIN {X 0,Y 403.418,Z 543.141,A -85,B 0,C 180,E1 -10889.001,E2 -10889.001} C_VEL
LIN {X 0,Y 403.48,Z 543.243,A -85,B 0,C 180,E1 -10890,E2 -10890} C_VEL
LIN {X 0,Y 403.442,Z 542.937,A -85,B 0,C 180,E1 -10890.998,E2 -10890.998} C_VEL
LIN {X 0,Y 403.418,Z 542.234,A -85,B 0,C 180,E1 -10891.996,E2 -10891.996} C_VEL
LIN {X 0,Y 403.455,Z 541.109,A -85,B 0,C 180,E1 -10892.995,E2 -10892.995} C_VEL
LIN {X 0,Y 403.378,Z 538.586,A -85,B 0,C 180,E1 -10894.496,E2 -10894.496} C_VEL
LIN {X 0,Y 403.332,Z 535.021,A -85,B 0,C 180,E1 -10896.001,E2 -10896.001} C_VEL
LIN {X 0,Y 403.27,Z 530.319,A -85,B 0,C 180,E1 -10897.51,E2 -10897.51} C_VEL
LIN {X 0,Y 403.384,Z 523.202,A -85,B 0,C 180,E1 -10899.274,E2 -10899.274} C_VEL
LIN {X 0,Y 403.693,Z 515.512,A -85,B 0,C 180,E1 -10900.786,E2 -10900.786} C_VEL
LIN {X 0,Y 404.074,Z 507.669,A -85,B 0,C 180,E1 -10902.046,E2 -10902.046} C_VEL
LIN {X 0,Y 404.682,Z 499.116,A -85,B 0,C 180,E1 -10903.187,E2 -10903.187} C_VEL
LIN {X 0,Y 405.388,Z 488.904,A -85,B 0,C 180,E1 -10904.302,E2 -10904.302} C_VEL
LIN {X 0,Y 406.156,Z 477.475,A -85,B 0,C 180,E1 -10905.3,E2 -10905.3} C_VEL
LIN {X 0,Y 406.971,Z 465.663,A -85,B 0,C 180,E1 -10906.103,E2 -10906.103} C_VEL
LIN {X 0,Y 407.724,Z 452.821,A -85,B 0,C 180,E1 -10906.748,E2 -10906.748} C_VEL
LIN {X 0,Y 408.255,Z 439.117,A -85,B 0,C 180,E1 -10907.209,E2 -10907.209} C_VEL
LIN {X 0,Y 408.714,Z 403.251,A -85,B 0,C 180,E1 -10907.867,E2 -10907.867} C_VEL
LIN {X 0,Y 409.048,Z 364.334,A -85,B 0,C 180,E1 -10908.548,E2 -10908.548} C_VEL
LIN {X 0,Y 405.143,Z 327.495,A -85,B 0,C 180,E1 -10909.375,E2 -10909.375} C_VEL
LIN {X 0,Y 405.986,Z 307.953,A -85,B 0,C 180,E1 -10912.385,E2 -10912.385} C_VEL
LIN {X 0,Y 407.216,Z 286.455,A -85,B 0,C 180,E1 -10915.749,E2 -10915.749} C_VEL
LIN {X 0,Y 407.861,Z 273.951,A -85,B 0,C 180,E1 -10917.725,E2 -10917.725} C_VEL
LIN {X 0,Y 405.428,Z 261.176,A -85,B 0,C 180,E1 -10919.918,E2 -10919.918} C_VEL
LIN {X 0,Y 404.176,Z 255.25,A -85,B 0,C 180,E1 -10921.005,E2 -10921.005} C_VEL
LIN {X 0,Y 404.133,Z 255.147,A -85,B 0,C 180,E1 -10923.812,E2 -10923.812} C_VEL
LIN {X 0,Y 404.124,Z 255.143,A -85,B 0,C 180,E1 -10926.872,E2 -10926.872} C_VEL
LIN {X 0,Y 404.111,Z 255.144,A -85,B 0,C 180,E1 -10930.074,E2 -10930.074} C_VEL
LIN {X 0,Y 404.133,Z 255.145,A -85,B 0,C 180,E1 -10933.081,E2 -10933.081} C_VEL
LIN {X 0,Y 404.112,Z 255.144,A -85,B 0,C 180,E1 -10935.921,E2 -10935.921} C_VEL
LIN {X 0,Y 404.093,Z 255.147,A -85,B 0,C 180,E1 -10938.632,E2 -10938.632} C_VEL
LIN {X 0,Y 404.129,Z 255.144,A -85,B 0,C 180,E1 -10941.494,E2 -10941.494} C_VEL
LIN {X 0,Y 404.161,Z 255.143,A -85,B 0,C 180,E1 -10944.982,E2 -10944.982} C_VEL
LIN {X 0,Y 404.121,Z 255.143,A -85,B 0,C 180,E1 -10948.444,E2 -10948.444} C_VEL
LIN {X 0,Y 404.137,Z 255.146,A -85,B 0,C 180,E1 -10950.861,E2 -10950.861} C_VEL
LIN {X 0,Y 404.14,Z 255.144,A -85,B 0,C 180,E1 -10954.723,E2 -10954.723} C_VEL
LIN {X 0,Y 404.154,Z 255.139,A -85,B 0,C 180,E1 -10957.507,E2 -10957.507} C_VEL
LIN {X 0,Y 404.149,Z 255.144,A -85,B 0,C 180,E1 -10960.707,E2 -10960.707} C_VEL
LIN {X 0,Y 404.204,Z 255.132,A -85,B 0,C 180,E1 -10963.848,E2 -10963.848} C_VEL
LIN {X 0,Y 404.272,Z 255.128,A -85,B 0,C 180,E1 -10966.939,E2 -10966.939} C_VEL
LIN {X 0,Y 404.235,Z 255.128,A -85,B 0,C 180,E1 -10969.988,E2 -10969.988} C_VEL
LIN {X 0,Y 404.323,Z 255.119,A -85,B 0,C 180,E1 -10973.011,E2 -10973.011} C_VEL
LIN {X 0,Y 404.243,Z 255.129,A -85,B 0,C 180,E1 -10975.013,E2 -10975.013} C_VEL
LIN {X 0,Y 404.461,Z 255.101,A -85,B 0,C 180,E1 -10978.009,E2 -10978.009} C_VEL
LIN {X 0,Y 404.456,Z 255.102,A -85,B 0,C 180,E1 -10981.992,E2 -10981.992} C_VEL
LIN {X 0,Y 404.323,Z 255.117,A -85,B 0,C 180,E1 -10986.616,E2 -10986.616} C_VEL
LIN {X 0,Y 404.242,Z 255.128,A -85,B 0,C 180,E1 -10989.002,E2 -10989.002} C_VEL
LIN {X 0,Y 404.235,Z 255.132,A -85,B 0,C 180,E1 -10992.042,E2 -10992.042} C_VEL
LIN {X 0,Y 404.188,Z 255.134,A -85,B 0,C 180,E1 -10995.119,E2 -10995.119} C_VEL
LIN {X 0,Y 404.192,Z 255.14,A -85,B 0,C 180,E1 -10998.239,E2 -10998.239} C_VEL
LIN {X 0,Y 404.127,Z 255.142,A -85,B 0,C 180,E1 -11001.42,E2 -11001.42} C_VEL
LIN {X 0,Y 404.125,Z 255.143,A -85,B 0,C 180,E1 -11004.669,E2 -11004.669} C_VEL
LIN {X 0,Y 404.094,Z 255.152,A -85,B 0,C 180,E1 -11008.008,E2 -11008.008} C_VEL
LIN {X 0,Y 404.133,Z 255.144,A -85,B 0,C 180,E1 -11010.287,E2 -11010.287} C_VEL
LIN {X 0,Y 404.129,Z 255.146,A -85,B 0,C 180,E1 -11013.814,E2 -11013.814} C_VEL
LIN {X 0,Y 404.123,Z 255.142,A -85,B 0,C 180,E1 -11016.875,E2 -11016.875} C_VEL
LIN {X 0,Y 404.111,Z 255.148,A -85,B 0,C 180,E1 -11020.076,E2 -11020.076} C_VEL
LIN {X 0,Y 404.135,Z 255.141,A -85,B 0,C 180,E1 -11023.083,E2 -11023.083} C_VEL
LIN {X 0,Y 404.114,Z 255.148,A -85,B 0,C 180,E1 -11025.923,E2 -11025.923} C_VEL
LIN {X 0,Y 404.095,Z 255.145,A -85,B 0,C 180,E1 -11028.634,E2 -11028.634} C_VEL
LIN {X 0,Y 404.132,Z 255.146,A -85,B 0,C 180,E1 -11031.497,E2 -11031.497} C_VEL
LIN {X 0,Y 404.168,Z 255.137,A -85,B 0,C 180,E1 -11034.984,E2 -11034.984} C_VEL
LIN {X 0,Y 404.128,Z 255.141,A -85,B 0,C 180,E1 -11038.446,E2 -11038.446} C_VEL
LIN {X 0,Y 404.146,Z 255.14,A -85,B 0,C 180,E1 -11040.863,E2 -11040.863} C_VEL
LIN {X 0,Y 404.151,Z 255.139,A -85,B 0,C 180,E1 -11044.724,E2 -11044.724} C_VEL
LIN {X 0,Y 404.165,Z 255.142,A -85,B 0,C 180,E1 -11047.509,E2 -11047.509} C_VEL
LIN {X 0,Y 404.14,Z 255.141,A -85,B 0,C 180,E1 -11050.707,E2 -11050.707} C_VEL
LIN {X 0,Y 404.174,Z 255.137,A -85,B 0,C 180,E1 -11053.847,E2 -11053.847} C_VEL
LIN {X 0,Y 404.267,Z 255.125,A -85,B 0,C 180,E1 -11056.939,E2 -11056.939} C_VEL
LIN {X 0,Y 404.244,Z 255.29,A -85,B 0,C 180,E1 -11058.912,E2 -11058.912} C_VEL
LIN {X 0,Y 404.469,Z 256.327,A -85,B 0,C 180,E1 -11059.082,E2 -11059.082} C_VEL
LIN {X 0,Y 409.958,Z 271.684,A -85,B 0,C 180,E1 -11059.606,E2 -11059.606} C_VEL
LIN {X 0,Y 409.106,Z 342.978,A -85,B 0,C 180,E1 -11060.872,E2 -11060.872} C_VEL
LIN {X 0,Y 408.985,Z 355.691,A -85,B 0,C 180,E1 -11061.291,E2 -11061.291} C_VEL
LIN {X 0,Y 408.649,Z 367.263,A -85,B 0,C 180,E1 -11061.844,E2 -11061.844} C_VEL
LIN {X 0,Y 408.248,Z 378.767,A -85,B 0,C 180,E1 -11062.582,E2 -11062.582} C_VEL
LIN {X 0,Y 407.693,Z 389.282,A -85,B 0,C 180,E1 -11063.443,E2 -11063.443} C_VEL
LIN {X 0,Y 407.026,Z 400.025,A -85,B 0,C 180,E1 -11064.551,E2 -11064.551} C_VEL
LIN {X 0,Y 406.42,Z 409.637,A -85,B 0,C 180,E1 -11065.786,E2 -11065.786} C_VEL
LIN {X 0,Y 405.82,Z 417.536,A -85,B 0,C 180,E1 -11067.022,E2 -11067.022} C_VEL
LIN {X 0,Y 405.187,Z 425.303,A -85,B 0,C 180,E1 -11068.51,E2 -11068.51} C_VEL
LIN {X 0,Y 404.741,Z 431.497,A -85,B 0,C 180,E1 -11070,E2 -11070} C_VEL
LIN {X 0,Y 404.392,Z 436.432,A -85,B 0,C 180,E1 -11071.494,E2 -11071.494} C_VEL
LIN {X 0,Y 404.03,Z 440.281,A -85,B 0,C 180,E1 -11072.992,E2 -11072.992} C_VEL
LIN {X 0,Y 403.925,Z 442.96,A -85,B 0,C 180,E1 -11074.444,E2 -11074.444} C_VEL
LIN {X 0,Y 403.267,Z 444.257,A -85,B 0,C 180,E1 -11075.258,E2 -11075.258} C_VEL
LIN {X 0,Y 400.352,Z 445.89,A -85,B 0,C 180,E1 -11076.59,E2 -11076.59} C_VEL
LIN {X 0,Y 397.433,Z 446.871,A -85,B 0,C 180,E1 -11077.951,E2 -11077.951} C_VEL
LIN {X 0,Y 396.785,Z 446.94,A -85,B 0,C 180,E1 -11078.802,E2 -11078.802} C_VEL
LIN {X 0,Y 396.885,Z 446.463,A -85,B 0,C 180,E1 -11080.2,E2 -11080.2} C_VEL
LIN {X 0,Y 397.16,Z 444.328,A -85,B 0,C 180,E1 -11082.26,E2 -11082.26} C_VEL
LIN {X 0,Y 397.419,Z 442.375,A -85,B 0,C 180,E1 -11083.434,E2 -11083.434} C_VEL
LIN {X 0,Y 397.918,Z 437.877,A -85,B 0,C 180,E1 -11085.363,E2 -11085.363} C_VEL
LIN {X 0,Y 398.476,Z 432.978,A -85,B 0,C 180,E1 -11086.919,E2 -11086.919} C_VEL
LIN {X 0,Y 399.167,Z 426.764,A -85,B 0,C 180,E1 -11088.477,E2 -11088.477} C_VEL
LIN {X 0,Y 400.019,Z 418.899,A -85,B 0,C 180,E1 -11090.035,E2 -11090.035} C_VEL
LIN {X 0,Y 400.841,Z 410.814,A -85,B 0,C 180,E1 -11091.334,E2 -11091.334} C_VEL
LIN {X 0,Y 401.671,Z 400.878,A -85,B 0,C 180,E1 -11092.639,E2 -11092.639} C_VEL
LIN {X 0,Y 402.487,Z 391.003,A -85,B 0,C 180,E1 -11093.679,E2 -11093.679} C_VEL
LIN {X 0,Y 403.273,Z 380.165,A -85,B 0,C 180,E1 -11094.587,E2 -11094.587} C_VEL
LIN {X 0,Y 403.832,Z 369.506,A -85,B 0,C 180,E1 -11095.293,E2 -11095.293} C_VEL
LIN {X 0,Y 404.198,Z 356.53,A -85,B 0,C 180,E1 -11095.938,E2 -11095.938} C_VEL
LIN {X 0,Y 404.368,Z 344.405,A -85,B 0,C 180,E1 -11096.342,E2 -11096.342} C_VEL
LIN {X 0,Y 404.814,Z 305.818,A -85,B 0,C 180,E1 -11097.064,E2 -11097.064} C_VEL
LIN {X 0,Y 405.224,Z 274.943,A -85,B 0,C 180,E1 -11097.623,E2 -11097.623} C_VEL
LIN {X 0,Y 397.292,Z 256.901,A -85,B 0,C 180,E1 -11098.492,E2 -11098.492} C_VEL
LIN {X 0,Y 397.133,Z 256.101,A -85,B 0,C 180,E1 -11098.687,E2 -11098.687} C_VEL
LIN {X 0,Y 397.078,Z 256.005,A -85,B 0,C 180,E1 -11102.071,E2 -11102.071} C_VEL
LIN {X 0,Y 397.1,Z 255.99,A -85,B 0,C 180,E1 -11105.498,E2 -11105.498} C_VEL
LIN {X 0,Y 397.092,Z 256.014,A -85,B 0,C 180,E1 -11108.854,E2 -11108.854} C_VEL
LIN {X 0,Y 397.054,Z 256.016,A -85,B 0,C 180,E1 -11112.268,E2 -11112.268} C_VEL
LIN {X 0,Y 397.083,Z 256.021,A -85,B 0,C 180,E1 -11115.069,E2 -11115.069} C_VEL
LIN {X 0,Y 397.05,Z 256.018,A -85,B 0,C 180,E1 -11118.023,E2 -11118.023} C_VEL
LIN {X 0,Y 397.087,Z 256.008,A -85,B 0,C 180,E1 -11121.723,E2 -11121.723} C_VEL
LIN {X 0,Y 397.122,Z 256.017,A -85,B 0,C 180,E1 -11125.506,E2 -11125.506} C_VEL
LIN {X 0,Y 397.074,Z 255.999,A -85,B 0,C 180,E1 -11129.117,E2 -11129.117} C_VEL
LIN {X 0,Y 397.075,Z 256.02,A -85,B 0,C 180,E1 -11132.246,E2 -11132.246} C_VEL
LIN {X 0,Y 397.114,Z 256.006,A -85,B 0,C 180,E1 -11135.98,E2 -11135.98} C_VEL
LIN {X 0,Y 397.135,Z 255.993,A -85,B 0,C 180,E1 -11139.704,E2 -11139.704} C_VEL
LIN {X 0,Y 397.178,Z 256.009,A -85,B 0,C 180,E1 -11142.844,E2 -11142.844} C_VEL
LIN {X 0,Y 397.224,Z 256.001,A -85,B 0,C 180,E1 -11146.702,E2 -11146.702} C_VEL
LIN {X 0,Y 397.207,Z 256.001,A -85,B 0,C 180,E1 -11149.808,E2 -11149.808} C_VEL
LIN {X 0,Y 397.286,Z 255.994,A -85,B 0,C 180,E1 -11152.887,E2 -11152.887} C_VEL
LIN {X 0,Y 397.22,Z 256,A -85,B 0,C 180,E1 -11154.924,E2 -11154.924} C_VEL
LIN {X 0,Y 397.432,Z 255.98,A -85,B 0,C 180,E1 -11157.973,E2 -11157.973} C_VEL
LIN {X 0,Y 397.436,Z 255.97,A -85,B 0,C 180,E1 -11162.027,E2 -11162.027} C_VEL
LIN {X 0,Y 397.308,Z 255.988,A -85,B 0,C 180,E1 -11166.092,E2 -11166.092} C_VEL
LIN {X 0,Y 397.228,Z 256,A -85,B 0,C 180,E1 -11169.162,E2 -11169.162} C_VEL
LIN {X 0,Y 397.211,Z 255.998,A -85,B 0,C 180,E1 -11172.258,E2 -11172.258} C_VEL
LIN {X 0,Y 397.168,Z 256.014,A -85,B 0,C 180,E1 -11175.392,E2 -11175.392} C_VEL
LIN {X 0,Y 397.151,Z 256.008,A -85,B 0,C 180,E1 -11178.574,E2 -11178.574} C_VEL
LIN {X 0,Y 397.088,Z 256.016,A -85,B 0,C 180,E1 -11181.819,E2 -11181.819} C_VEL
LIN {X 0,Y 397.097,Z 256.019,A -85,B 0,C 180,E1 -11185.136,E2 -11185.136} C_VEL
LIN {X 0,Y 397.056,Z 256.011,A -85,B 0,C 180,E1 -11188.549,E2 -11188.549} C_VEL
LIN {X 0,Y 397.072,Z 256.02,A -85,B 0,C 180,E1 -11191.835,E2 -11191.835} C_VEL
LIN {X 0,Y 397.114,Z 256.006,A -85,B 0,C 180,E1 -11194.494,E2 -11194.494} C_VEL
LIN {X 0,Y 397.085,Z 256.016,A -85,B 0,C 180,E1 -11198.277,E2 -11198.277} C_VEL
LIN {X 0,Y 397.047,Z 256.026,A -85,B 0,C 180,E1 -11201.977,E2 -11201.977} C_VEL
LIN {X 0,Y 397.082,Z 256.024,A -85,B 0,C 180,E1 -11205.07,E2 -11205.07} C_VEL
LIN {X 0,Y 397.048,Z 256.027,A -85,B 0,C 180,E1 -11208.024,E2 -11208.024} C_VEL
LIN {X 0,Y 397.085,Z 256.009,A -85,B 0,C 180,E1 -11211.724,E2 -11211.724} C_VEL
LIN {X 0,Y 397.114,Z 256.007,A -85,B 0,C 180,E1 -11215.506,E2 -11215.506} C_VEL
LIN {X 0,Y 397.14,Z 256.258,A -85,B 0,C 180,E1 -11217.428,E2 -11217.428} C_VEL
LIN {X 0,Y 400.278,Z 269.465,A -85,B 0,C 180,E1 -11220.008,E2 -11220.008} C_VEL
LIN {X 0,Y 402.097,Z 278.254,A -85,B 0,C 180,E1 -11221.639,E2 -11221.639} C_VEL
LIN {X 0,Y 400.872,Z 295.977,A -85,B 0,C 180,E1 -11224.562,E2 -11224.562} C_VEL
LIN {X 0,Y 399.267,Z 319.037,A -85,B 0,C 180,E1 -11228.306,E2 -11228.306} C_VEL
LIN {X 0,Y 398.937,Z 325.466,A -85,B 0,C 180,E1 -11229.312,E2 -11229.312} C_VEL
LIN {X 0,Y 400.748,Z 337.857,A -85,B 0,C 180,E1 -11229.691,E2 -11229.691} C_VEL
LIN {X 0,Y 403.688,Z 362.057,A -85,B 0,C 180,E1 -11230.314,E2 -11230.314} C_VEL
LIN {X 0,Y 404.129,Z 368.113,A -85,B 0,C 180,E1 -11230.452,E2 -11230.452} C_VEL
LIN {X 0,Y 403.096,Z 436.77,A -85,B 0,C 180,E1 -11231.71,E2 -11231.71} C_VEL
LIN {X 0,Y 402.437,Z 450.602,A -85,B 0,C 180,E1 -11232.172,E2 -11232.172} C_VEL
LIN {X 0,Y 401.456,Z 463.561,A -85,B 0,C 180,E1 -11232.817,E2 -11232.817} C_VEL
LIN {X 0,Y 400.504,Z 474.583,A -85,B 0,C 180,E1 -11233.563,E2 -11233.563} C_VEL
LIN {X 0,Y 399.417,Z 486.148,A -85,B 0,C 180,E1 -11234.566,E2 -11234.566} C_VEL
LIN {X 0,Y 398.454,Z 496.614,A -85,B 0,C 180,E1 -11235.704,E2 -11235.704} C_VEL
LIN {X 0,Y 397.709,Z 506.088,A -85,B 0,C 180,E1 -11236.979,E2 -11236.979} C_VEL
LIN {X 0,Y 396.991,Z 513.9,A -85,B 0,C 180,E1 -11238.253,E2 -11238.253} C_VEL
LIN {X 0,Y 396.398,Z 521.591,A -85,B 0,C 180,E1 -11239.787,E2 -11239.787} C_VEL
LIN {X 0,Y 396.175,Z 527.833,A -85,B 0,C 180,E1 -11241.327,E2 -11241.327} C_VEL
LIN {X 0,Y 396.099,Z 532.815,A -85,B 0,C 180,E1 -11242.865,E2 -11242.865} C_VEL
LIN {X 0,Y 396.162,Z 536.676,A -85,B 0,C 180,E1 -11244.4,E2 -11244.4} C_VEL
LIN {X 0,Y 396.292,Z 539.511,A -85,B 0,C 180,E1 -11245.932,E2 -11245.932} C_VEL
LIN {X 0,Y 396.382,Z 540.863,A -85,B 0,C 180,E1 -11246.951,E2 -11246.951} C_VEL
LIN {X 0,Y 396.323,Z 541.795,A -85,B 0,C 180,E1 -11247.967,E2 -11247.967} C_VEL
LIN {X 0,Y 396.364,Z 542.297,A -85,B 0,C 180,E1 -11248.984,E2 -11248.984} C_VEL
LIN {X 0,Y 396.431,Z 542.388,A -85,B 0,C 180,E1 -11250,E2 -11250} C_VEL
LIN {X 0,Y 396.391,Z 542.069,A -85,B 0,C 180,E1 -11251.015,E2 -11251.015} C_VEL
LIN {X 0,Y 396.366,Z 541.353,A -85,B 0,C 180,E1 -11252.032,E2 -11252.032} C_VEL
LIN {X 0,Y 396.407,Z 540.203,A -85,B 0,C 180,E1 -11253.048,E2 -11253.048} C_VEL
LIN {X 0,Y 396.313,Z 537.654,A -85,B 0,C 180,E1 -11254.577,E2 -11254.577} C_VEL
LIN {X 0,Y 396.248,Z 534.058,A -85,B 0,C 180,E1 -11256.108,E2 -11256.108} C_VEL
LIN {X 0,Y 396.186,Z 529.319,A -85,B 0,C 180,E1 -11257.645,E2 -11257.645} C_VEL
LIN {X 0,Y 396.287,Z 523.31,A -85,B 0,C 180,E1 -11259.184,E2 -11259.184} C_VEL
LIN {X 0,Y 396.602,Z 515.822,A -85,B 0,C 180,E1 -11260.723,E2 -11260.723} C_VEL
LIN {X 0,Y 397.086,Z 506.542,A -85,B 0,C 180,E1 -11262.262,E2 -11262.262} C_VEL
LIN {X 0,Y 397.735,Z 496.949,A -85,B 0,C 180,E1 -11263.538,E2 -11263.538} C_VEL
LIN {X 0,Y 398.483,Z 486.287,A -85,B 0,C 180,E1 -11264.686,E2 -11264.686} C_VEL
LIN {X 0,Y 399.402,Z 474.481,A -85,B 0,C 180,E1 -11265.696,E2 -11265.696} C_VEL
LIN {X 0,Y 400.171,Z 463.028,A -85,B 0,C 180,E1 -11266.45,E2 -11266.45} C_VEL
LIN {X 0,Y 400.964,Z 449.395,A -85,B 0,C 180,E1 -11267.105,E2 -11267.105} C_VEL
LIN {X 0,Y 401.478,Z 436.714,A -85,B 0,C 180,E1 -11267.509,E2 -11267.509} C_VEL
LIN {X 0,Y 402.192,Z 364.856,A -85,B 0,C 180,E1 -11268.807,E2 -11268.807} C_VEL
LIN {X 0,Y 398.163,Z 326.466,A -85,B 0,C 180,E1 -11269.695,E2 -11269.695} C_VEL
LIN {X 0,Y 399.17,Z 305.092,A -85,B 0,C 180,E1 -11273.062,E2 -11273.062} C_VEL
LIN {X 0,Y 400.41,Z 284.484,A -85,B 0,C 180,E1 -11276.349,E2 -11276.349} C_VEL
LIN {X 0,Y 400.857,Z 274.454,A -85,B 0,C 180,E1 -11277.968,E2 -11277.968} C_VEL
LIN {X 0,Y 397.55,Z 258.172,A -85,B 0,C 180,E1 -11280.841,E2 -11280.841} C_VEL
LIN {X 0,Y 397.121,Z 256.131,A -85,B 0,C 180,E1 -11281.247,E2 -11281.247} C_VEL
LIN {X 0,Y 397.111,Z 256.02,A -85,B 0,C 180,E1 -11284.493,E2 -11284.493} C_VEL
LIN {X 0,Y 397.08,Z 256.019,A -85,B 0,C 180,E1 -11288.276,E2 -11288.276} C_VEL
LIN {X 0,Y 397.043,Z 256.024,A -85,B 0,C 180,E1 -11291.975,E2 -11291.975} C_VEL
LIN {X 0,Y 397.077,Z 256.024,A -85,B 0,C 180,E1 -11295.068,E2 -11295.068} C_VEL
LIN {X 0,Y 397.042,Z 256.024,A -85,B 0,C 180,E1 -11298.023,E2 -11298.023} C_VEL
LIN {X 0,Y 397.081,Z 256.02,A -85,B 0,C 180,E1 -11301.723,E2 -11301.723} C_VEL
LIN {X 0,Y 397.105,Z 256.018,A -85,B 0,C 180,E1 -11305.505,E2 -11305.505} C_VEL
LIN {X 0,Y 397.062,Z 256.027,A -85,B 0,C 180,E1 -11309.116,E2 -11309.116} C_VEL
LIN {X 0,Y 397.047,Z 256.024,A -85,B 0,C 180,E1 -11312.252,E2 -11312.252} C_VEL
LIN {X 0,Y 397.09,Z 256.024,A -85,B 0,C 180,E1 -11314.864,E2 -11314.864} C_VEL
LIN {X 0,Y 397.082,Z 256.02,A -85,B 0,C 180,E1 -11318.181,E2 -11318.181} C_VEL
LIN {X 0,Y 397.144,Z 256.012,A -85,B 0,C 180,E1 -11321.426,E2 -11321.426} C_VEL
LIN {X 0,Y 397.16,Z 256.014,A -85,B 0,C 180,E1 -11324.607,E2 -11324.607} C_VEL
LIN {X 0,Y 397.205,Z 256.003,A -85,B 0,C 180,E1 -11327.742,E2 -11327.742} C_VEL
LIN {X 0,Y 397.216,Z 256.007,A -85,B 0,C 180,E1 -11330.837,E2 -11330.837} C_VEL
LIN {X 0,Y 397.302,Z 255.992,A -85,B 0,C 180,E1 -11333.908,E2 -11333.908} C_VEL
LIN {X 0,Y 397.43,Z 255.977,A -85,B 0,C 180,E1 -11337.973,E2 -11337.973} C_VEL
LIN {X 0,Y 397.423,Z 255.979,A -85,B 0,C 180,E1 -11342.027,E2 -11342.027} C_VEL
LIN {X 0,Y 397.277,Z 255.994,A -85,B 0,C 180,E1 -11346.613,E2 -11346.613} C_VEL
LIN {X 0,Y 397.213,Z 256.003,A -85,B 0,C 180,E1 -11349.163,E2 -11349.163} C_VEL
LIN {X 0,Y 397.201,Z 256.011,A -85,B 0,C 180,E1 -11352.259,E2 -11352.259} C_VEL
LIN {X 0,Y 397.162,Z 256.009,A -85,B 0,C 180,E1 -11355.393,E2 -11355.393} C_VEL
LIN {X 0,Y 397.146,Z 256.014,A -85,B 0,C 180,E1 -11358.575,E2 -11358.575} C_VEL
LIN {X 0,Y 397.084,Z 256.022,A -85,B 0,C 180,E1 -11361.82,E2 -11361.82} C_VEL
LIN {X 0,Y 397.093,Z 256.017,A -85,B 0,C 180,E1 -11365.136,E2 -11365.136} C_VEL
LIN {X 0,Y 397.053,Z 256.024,A -85,B 0,C 180,E1 -11368.549,E2 -11368.549} C_VEL
LIN {X 0,Y 397.071,Z 256.025,A -85,B 0,C 180,E1 -11371.837,E2 -11371.837} C_VEL
LIN {X 0,Y 397.108,Z 256.017,A -85,B 0,C 180,E1 -11374.496,E2 -11374.496} C_VEL
LIN {X 0,Y 397.081,Z 256.022,A -85,B 0,C 180,E1 -11378.278,E2 -11378.278} C_VEL
LIN {X 0,Y 397.044,Z 256.029,A -85,B 0,C 180,E1 -11381.977,E2 -11381.977} C_VEL
LIN {X 0,Y 397.078,Z 256.02,A -85,B 0,C 180,E1 -11385.071,E2 -11385.071} C_VEL
LIN {X 0,Y 397.045,Z 256.027,A -85,B 0,C 180,E1 -11388.025,E2 -11388.025} C_VEL
LIN {X 0,Y 397.085,Z 256.025,A -85,B 0,C 180,E1 -11391.725,E2 -11391.725} C_VEL
LIN {X 0,Y 397.112,Z 256.021,A -85,B 0,C 180,E1 -11395.507,E2 -11395.507} C_VEL
LIN {X 0,Y 397.069,Z 256.023,A -85,B 0,C 180,E1 -11399.118,E2 -11399.118} C_VEL
LIN {X 0,Y 397.057,Z 256.022,A -85,B 0,C 180,E1 -11402.254,E2 -11402.254} C_VEL
LIN {X 0,Y 397.1,Z 256.018,A -85,B 0,C 180,E1 -11404.866,E2 -11404.866} C_VEL
LIN {X 0,Y 397.091,Z 256.018,A -85,B 0,C 180,E1 -11408.182,E2 -11408.182} C_VEL
LIN {X 0,Y 397.1,Z 256.022,A -85,B 0,C 180,E1 -11411.424,E2 -11411.424} C_VEL
LIN {X 0,Y 397.124,Z 256.018,A -85,B 0,C 180,E1 -11413.552,E2 -11413.552} C_VEL
LIN {X 0,Y 397.193,Z 256.005,A -85,B 0,C 180,E1 -11416.702,E2 -11416.702} C_VEL
LIN {X 0,Y 397.208,Z 256.121,A -85,B 0,C 180,E1 -11418.584,E2 -11418.584} C_VEL
LIN {X 0,Y 397.381,Z 257.015,A -85,B 0,C 180,E1 -11418.766,E2 -11418.766} C_VEL
LIN {X 0,Y 403.073,Z 272.551,A -85,B 0,C 180,E1 -11419.326,E2 -11419.326} C_VEL
LIN {X 0,Y 402.297,Z 343.48,A -85,B 0,C 180,E1 -11420.608,E2 -11420.608} C_VEL
LIN {X 0,Y 402.163,Z 355.893,A -85,B 0,C 180,E1 -11421.015,E2 -11421.015} C_VEL
LIN {X 0,Y 401.813,Z 367.63,A -85,B 0,C 180,E1 -11421.577,E2 -11421.577} C_VEL
LIN {X 0,Y 401.4,Z 379.235,A -85,B 0,C 180,E1 -11422.328,E2 -11422.328} C_VEL
LIN {X 0,Y 400.821,Z 389.823,A -85,B 0,C 180,E1 -11423.203,E2 -11423.203} C_VEL
LIN {X 0,Y 400.142,Z 400.637,A -85,B 0,C 180,E1 -11424.331,E2 -11424.331} C_VEL
LIN {X 0,Y 399.439,Z 411.164,A -85,B 0,C 180,E1 -11425.712,E2 -11425.712} C_VEL
LIN {X 0,Y 398.818,Z 418.952,A -85,B 0,C 180,E1 -11426.97,E2 -11426.97} C_VEL
LIN {X 0,Y 398.15,Z 426.592,A -85,B 0,C 180,E1 -11428.483,E2 -11428.483} C_VEL
LIN {X 0,Y 397.714,Z 432.691,A -85,B 0,C 180,E1 -11430,E2 -11430} C_VEL
LIN {X 0,Y 397.336,Z 437.555,A -85,B 0,C 180,E1 -11431.521,E2 -11431.521} C_VEL
LIN {X 0,Y 396.974,Z 441.336,A -85,B 0,C 180,E1 -11433.045,E2 -11433.045} C_VEL
LIN {X 0,Y 396.875,Z 443.813,A -85,B 0,C 180,E1 -11434.42,E2 -11434.42} C_VEL
LIN {X 0,Y 396.826,Z 445.924,A -85,B 0,C 180,E1 -11436.1,E2 -11436.1} C_VEL
LIN {X 0,Y 396.778,Z 446.967,A -85,B 0,C 180,E1 -11438.147,E2 -11438.147} C_VEL
LIN {X 0,Y 396.785,Z 446.94,A -85,B 0,C 180,E1 -11438.802,E2 -11438.802} C_VEL
LIN {X 0,Y 396.176,Z 446.847,A -85,B 0,C 180,E1 -11439.65,E2 -11439.65} C_VEL
LIN {X 0,Y 393.46,Z 446.278,A -85,B 0,C 180,E1 -11441.03,E2 -11441.03} C_VEL
LIN {X 0,Y 391.222,Z 445.347,A -85,B 0,C 180,E1 -11442.137,E2 -11442.137} C_VEL
LIN {X 0,Y 390.366,Z 444.248,A -85,B 0,C 180,E1 -11442.981,E2 -11442.981} C_VEL
LIN {X 0,Y 390.353,Z 443.755,A -85,B 0,C 180,E1 -11443.264,E2 -11443.264} C_VEL
LIN {X 0,Y 390.829,Z 439.861,A -85,B 0,C 180,E1 -11445.114,E2 -11445.114} C_VEL
LIN {X 0,Y 391.387,Z 435.277,A -85,B 0,C 180,E1 -11446.697,E2 -11446.697} C_VEL
LIN {X 0,Y 392.112,Z 429.173,A -85,B 0,C 180,E1 -11448.338,E2 -11448.338} C_VEL
LIN {X 0,Y 392.988,Z 422.039,A -85,B 0,C 180,E1 -11449.864,E2 -11449.864} C_VEL
LIN {X 0,Y 393.775,Z 414.478,A -85,B 0,C 180,E1 -11451.185,E2 -11451.185} C_VEL
LIN {X 0,Y 394.724,Z 405.211,A -85,B 0,C 180,E1 -11452.507,E2 -11452.507} C_VEL
LIN {X 0,Y 395.51,Z 396.094,A -85,B 0,C 180,E1 -11453.566,E2 -11453.566} C_VEL
LIN {X 0,Y 396.199,Z 386.334,A -85,B 0,C 180,E1 -11454.496,E2 -11454.496} C_VEL
LIN {X 0,Y 396.874,Z 374.964,A -85,B 0,C 180,E1 -11455.355,E2 -11455.355} C_VEL
LIN {X 0,Y 397.5,Z 361.952,A -85,B 0,C 180,E1 -11456.091,E2 -11456.091} C_VEL
LIN {X 0,Y 397.703,Z 349.287,A -85,B 0,C 180,E1 -11456.589,E2 -11456.589} C_VEL
LIN {X 0,Y 397.878,Z 333.335,A -85,B 0,C 180,E1 -11456.948,E2 -11456.948} C_VEL
LIN {X 0,Y 398.729,Z 276.891,A -85,B 0,C 180,E1 -11457.982,E2 -11457.982} C_VEL
LIN {X 0,Y 390.354,Z 258.134,A -85,B 0,C 180,E1 -11458.906,E2 -11458.906} C_VEL
LIN {X 0,Y 390.12,Z 257.197,A -85,B 0,C 180,E1 -11459.039,E2 -11459.039} C_VEL
LIN {X 0,Y 390.074,Z 256.882,A -85,B 0,C 180,E1 -11459.701,E2 -11459.701} C_VEL
LIN {X 0,Y 390.043,Z 256.892,A -85,B 0,C 180,E1 -11462.721,E2 -11462.721} C_VEL
LIN {X 0,Y 390.043,Z 256.864,A -85,B 0,C 180,E1 -11465.822,E2 -11465.822} C_VEL
LIN {X 0,Y 390.037,Z 256.9,A -85,B 0,C 180,E1 -11469.212,E2 -11469.212} C_VEL
LIN {X 0,Y 390.03,Z 256.891,A -85,B 0,C 180,E1 -11472.371,E2 -11472.371} C_VEL
LIN {X 0,Y 390.039,Z 256.897,A -85,B 0,C 180,E1 -11475.353,E2 -11475.353} C_VEL
LIN {X 0,Y 390.013,Z 256.895,A -85,B 0,C 180,E1 -11478.184,E2 -11478.184} C_VEL
LIN {X 0,Y 390.054,Z 256.89,A -85,B 0,C 180,E1 -11480.903,E2 -11480.903} C_VEL
LIN {X 0,Y 390.081,Z 256.896,A -85,B 0,C 180,E1 -11484.792,E2 -11484.792} C_VEL
LIN {X 0,Y 390.02,Z 256.882,A -85,B 0,C 180,E1 -11488.495,E2 -11488.495} C_VEL
LIN {X 0,Y 390.021,Z 256.896,A -85,B 0,C 180,E1 -11492.062,E2 -11492.062} C_VEL
LIN {X 0,Y 390.044,Z 256.895,A -85,B 0,C 180,E1 -11495.517,E2 -11495.517} C_VEL
LIN {X 0,Y 390.051,Z 256.868,A -85,B 0,C 180,E1 -11498.877,E2 -11498.877} C_VEL
LIN {X 0,Y 390.123,Z 256.891,A -85,B 0,C 180,E1 -11502.166,E2 -11502.166} C_VEL
LIN {X 0,Y 390.137,Z 256.879,A -85,B 0,C 180,E1 -11505.392,E2 -11505.392} C_VEL
LIN {X 0,Y 390.139,Z 256.885,A -85,B 0,C 180,E1 -11508.571,E2 -11508.571} C_VEL
LIN {X 0,Y 390.25,Z 256.872,A -85,B 0,C 180,E1 -11512.087,E2 -11512.087} C_VEL
LIN {X 0,Y 390.192,Z 256.876,A -85,B 0,C 180,E1 -11514.833,E2 -11514.833} C_VEL
LIN {X 0,Y 390.399,Z 256.856,A -85,B 0,C 180,E1 -11517.936,E2 -11517.936} C_VEL
LIN {X 0,Y 390.403,Z 256.845,A -85,B 0,C 180,E1 -11522.063,E2 -11522.063} C_VEL
LIN {X 0,Y 390.264,Z 256.865,A -85,B 0,C 180,E1 -11526.203,E2 -11526.203} C_VEL
LIN {X 0,Y 390.185,Z 256.879,A -85,B 0,C 180,E1 -11529.329,E2 -11529.329} C_VEL
LIN {X 0,Y 390.164,Z 256.875,A -85,B 0,C 180,E1 -11532.483,E2 -11532.483} C_VEL
LIN {X 0,Y 390.13,Z 256.889,A -85,B 0,C 180,E1 -11535.677,E2 -11535.677} C_VEL
LIN {X 0,Y 390.096,Z 256.889,A -85,B 0,C 180,E1 -11538.922,E2 -11538.922} C_VEL
LIN {X 0,Y 390.029,Z 256.895,A -85,B 0,C 180,E1 -11542.235,E2 -11542.235} C_VEL
LIN {X 0,Y 390.045,Z 256.891,A -85,B 0,C 180,E1 -11545.722,E2 -11545.722} C_VEL
LIN {X 0,Y 390.018,Z 256.894,A -85,B 0,C 180,E1 -11549.113,E2 -11549.113} C_VEL
LIN {X 0,Y 390.035,Z 256.892,A -85,B 0,C 180,E1 -11552.722,E2 -11552.722} C_VEL
LIN {X 0,Y 390.047,Z 256.898,A -85,B 0,C 180,E1 -11555.825,E2 -11555.825} C_VEL
LIN {X 0,Y 390.031,Z 256.893,A -85,B 0,C 180,E1 -11559.212,E2 -11559.212} C_VEL
LIN {X 0,Y 390.026,Z 256.9,A -85,B 0,C 180,E1 -11562.372,E2 -11562.372} C_VEL
LIN {X 0,Y 390.037,Z 256.899,A -85,B 0,C 180,E1 -11565.354,E2 -11565.354} C_VEL
LIN {X 0,Y 390.011,Z 256.905,A -85,B 0,C 180,E1 -11568.185,E2 -11568.185} C_VEL
LIN {X 0,Y 390.053,Z 256.877,A -85,B 0,C 180,E1 -11570.904,E2 -11570.904} C_VEL
LIN {X 0,Y 390.066,Z 256.882,A -85,B 0,C 180,E1 -11574.792,E2 -11574.792} C_VEL
LIN {X 0,Y 390.114,Z 257.067,A -85,B 0,C 180,E1 -11577.017,E2 -11577.017} C_VEL
LIN {X 0,Y 393.391,Z 270.875,A -85,B 0,C 180,E1 -11579.782,E2 -11579.782} C_VEL
LIN {X 0,Y 395.287,Z 280.526,A -85,B 0,C 180,E1 -11581.602,E2 -11581.602} C_VEL
LIN {X 0,Y 393.807,Z 298.693,A -85,B 0,C 180,E1 -11584.64,E2 -11584.64} C_VEL
LIN {X 0,Y 392.322,Z 320.004,A -85,B 0,C 180,E1 -11588.162,E2 -11588.162} C_VEL
LIN {X 0,Y 392.087,Z 324.724,A -85,B 0,C 180,E1 -11588.894,E2 -11588.894} C_VEL
LIN {X 0,Y 395.74,Z 350.409,A -85,B 0,C 180,E1 -11589.639,E2 -11589.639} C_VEL
LIN {X 0,Y 397.537,Z 367.814,A -85,B 0,C 180,E1 -11590.077,E2 -11590.077} C_VEL
LIN {X 0,Y 396.474,Z 435.596,A -85,B 0,C 180,E1 -11591.336,E2 -11591.336} C_VEL
LIN {X 0,Y 395.78,Z 449.3,A -85,B 0,C 180,E1 -11591.795,E2 -11591.795} C_VEL
LIN {X 0,Y 394.758,Z 462.398,A -85,B 0,C 180,E1 -11592.45,E2 -11592.45} C_VEL
LIN {X 0,Y 393.676,Z 474.275,A -85,B 0,C 180,E1 -11593.27,E2 -11593.27} C_VEL
LIN {X 0,Y 392.558,Z 485.735,A -85,B 0,C 180,E1 -11594.289,E2 -11594.289} C_VEL
LIN {X 0,Y 391.516,Z 496.117,A -85,B 0,C 180,E1 -11595.445,E2 -11595.445} C_VEL
LIN {X 0,Y 390.763,Z 505.505,A -85,B 0,C 180,E1 -11596.743,E2 -11596.743} C_VEL
LIN {X 0,Y 389.989,Z 513.266,A -85,B 0,C 180,E1 -11598.039,E2 -11598.039} C_VEL
LIN {X 0,Y 389.359,Z 520.915,A -85,B 0,C 180,E1 -11599.601,E2 -11599.601} C_VEL
LIN {X 0,Y 389.12,Z 527.121,A -85,B 0,C 180,E1 -11601.169,E2 -11601.169} C_VEL
LIN {X 0,Y 389.02,Z 532.071,A -85,B 0,C 180,E1 -11602.735,E2 -11602.735} C_VEL
LIN {X 0,Y 389.1,Z 535.906,A -85,B 0,C 180,E1 -11604.298,E2 -11604.298} C_VEL
LIN {X 0,Y 389.227,Z 538.715,A -85,B 0,C 180,E1 -11605.858,E2 -11605.858} C_VEL
LIN {X 0,Y 389.332,Z 540.057,A -85,B 0,C 180,E1 -11606.895,E2 -11606.895} C_VEL
LIN {X 0,Y 389.269,Z 540.972,A -85,B 0,C 180,E1 -11607.93,E2 -11607.93} C_VEL
LIN {X 0,Y 389.311,Z 541.452,A -85,B 0,C 180,E1 -11608.965,E2 -11608.965} C_VEL
LIN {X 0,Y 389.382,Z 541.531,A -85,B 0,C 180,E1 -11610,E2 -11610} C_VEL
LIN {X 0,Y 389.34,Z 541.2,A -85,B 0,C 180,E1 -11611.034,E2 -11611.034} C_VEL
LIN {X 0,Y 389.315,Z 540.47,A -85,B 0,C 180,E1 -11612.069,E2 -11612.069} C_VEL
LIN {X 0,Y 389.36,Z 539.294,A -85,B 0,C 180,E1 -11613.104,E2 -11613.104} C_VEL
LIN {X 0,Y 389.25,Z 536.715,A -85,B 0,C 180,E1 -11614.66,E2 -11614.66} C_VEL
LIN {X 0,Y 389.143,Z 531.928,A -85,B 0,C 180,E1 -11616.63,E2 -11616.63} C_VEL
LIN {X 0,Y 389.15,Z 526.447,A -85,B 0,C 180,E1 -11618.306,E2 -11618.306} C_VEL
LIN {X 0,Y 389.301,Z 519.956,A -85,B 0,C 180,E1 -11619.874,E2 -11619.874} C_VEL
LIN {X 0,Y 389.712,Z 511.841,A -85,B 0,C 180,E1 -11621.441,E2 -11621.441} C_VEL
LIN {X 0,Y 390.302,Z 503.597,A -85,B 0,C 180,E1 -11622.742,E2 -11622.742} C_VEL
LIN {X 0,Y 390.96,Z 493.976,A -85,B 0,C 180,E1 -11623.991,E2 -11623.991} C_VEL
LIN {X 0,Y 391.639,Z 483.664,A -85,B 0,C 180,E1 -11625.081,E2 -11625.081} C_VEL
LIN {X 0,Y 392.549,Z 473.046,A -85,B 0,C 180,E1 -11625.977,E2 -11625.977} C_VEL
LIN {X 0,Y 393.32,Z 461.379,A -85,B 0,C 180,E1 -11626.745,E2 -11626.745} C_VEL
LIN {X 0,Y 394.132,Z 448.244,A -85,B 0,C 180,E1 -11627.377,E2 -11627.377} C_VEL
LIN {X 0,Y 394.632,Z 435.33,A -85,B 0,C 180,E1 -11627.79,E2 -11627.79} C_VEL
LIN {X 0,Y 395.285,Z 364.845,A -85,B 0,C 180,E1 -11629.084,E2 -11629.084} C_VEL
LIN {X 0,Y 391.211,Z 325.661,A -85,B 0,C 180,E1 -11630.008,E2 -11630.008} C_VEL
LIN {X 0,Y 392.263,Z 304.187,A -85,B 0,C 180,E1 -11633.446,E2 -11633.446} C_VEL
LIN {X 0,Y 393.458,Z 285.247,A -85,B 0,C 180,E1 -11636.522,E2 -11636.522} C_VEL
LIN {X 0,Y 393.987,Z 276.708,A -85,B 0,C 180,E1 -11637.92,E2 -11637.92} C_VEL
LIN {X 0,Y 391.309,Z 262.537,A -85,B 0,C 180,E1 -11640.448,E2 -11640.448} C_VEL
LIN {X 0,Y 390.055,Z 257.014,A -85,B 0,C 180,E1 -11641.5,E2 -11641.5} C_VEL
LIN {X 0,Y 390.063,Z 256.899,A -85,B 0,C 180,E1 -11645.208,E2 -11645.208} C_VEL
LIN {X 0,Y 390.047,Z 256.899,A -85,B 0,C 180,E1 -11649.096,E2 -11649.096} C_VEL
LIN {X 0,Y 390.022,Z 256.898,A -85,B 0,C 180,E1 -11652.371,E2 -11652.371} C_VEL
LIN {X 0,Y 390.033,Z 256.903,A -85,B 0,C 180,E1 -11655.353,E2 -11655.353} C_VEL
LIN {X 0,Y 390.006,Z 256.9,A -85,B 0,C 180,E1 -11658.183,E2 -11658.183} C_VEL
LIN {X 0,Y 390.048,Z 256.899,A -85,B 0,C 180,E1 -11660.903,E2 -11660.903} C_VEL
LIN {X 0,Y 390.058,Z 256.897,A -85,B 0,C 180,E1 -11664.79,E2 -11664.79} C_VEL
LIN {X 0,Y 390.007,Z 256.902,A -85,B 0,C 180,E1 -11668.494,E2 -11668.494} C_VEL
LIN {X 0,Y 390.005,Z 256.9,A -85,B 0,C 180,E1 -11672.002,E2 -11672.002} C_VEL
LIN {X 0,Y 390.03,Z 256.898,A -85,B 0,C 180,E1 -11675.516,E2 -11675.516} C_VEL
LIN {X 0,Y 390.041,Z 256.903,A -85,B 0,C 180,E1 -11678.877,E2 -11678.877} C_VEL
LIN {X 0,Y 390.099,Z 256.89,A -85,B 0,C 180,E1 -11682.165,E2 -11682.165} C_VEL
LIN {X 0,Y 390.127,Z 256.886,A -85,B 0,C 180,E1 -11685.392,E2 -11685.392} C_VEL
LIN {X 0,Y 390.13,Z 256.89,A -85,B 0,C 180,E1 -11688.571,E2 -11688.571} C_VEL
LIN {X 0,Y 390.244,Z 256.872,A -85,B 0,C 180,E1 -11692.087,E2 -11692.087} C_VEL
LIN {X 0,Y 390.185,Z 256.882,A -85,B 0,C 180,E1 -11694.833,E2 -11694.833} C_VEL
LIN {X 0,Y 390.397,Z 256.853,A -85,B 0,C 180,E1 -11697.937,E2 -11697.937} C_VEL
LIN {X 0,Y 390.389,Z 256.855,A -85,B 0,C 180,E1 -11702.064,E2 -11702.064} C_VEL
LIN {X 0,Y 390.236,Z 256.873,A -85,B 0,C 180,E1 -11706.607,E2 -11706.607} C_VEL
LIN {X 0,Y 390.172,Z 256.88,A -85,B 0,C 180,E1 -11709.33,E2 -11709.33} C_VEL
LIN {X 0,Y 390.184,Z 256.878,A -85,B 0,C 180,E1 -11713.439,E2 -11713.439} C_VEL
LIN {X 0,Y 390.119,Z 256.886,A -85,B 0,C 180,E1 -11717.299,E2 -11717.299} C_VEL
LIN {X 0,Y 390.078,Z 256.895,A -85,B 0,C 180,E1 -11720.471,E2 -11720.471} C_VEL
LIN {X 0,Y 390.047,Z 256.896,A -85,B 0,C 180,E1 -11723.354,E2 -11723.354} C_VEL
LIN {X 0,Y 390.02,Z 256.899,A -85,B 0,C 180,E1 -11726.776,E2 -11726.776} C_VEL
LIN {X 0,Y 390.027,Z 256.901,A -85,B 0,C 180,E1 -11730.301,E2 -11730.301} C_VEL
LIN {X 0,Y 390.061,Z 256.899,A -85,B 0,C 180,E1 -11734.026,E2 -11734.026} C_VEL
LIN {X 0,Y 390.028,Z 256.903,A -85,B 0,C 180,E1 -11737.782,E2 -11737.782} C_VEL
LIN {X 0,Y 390.009,Z 256.9,A -85,B 0,C 180,E1 -11740.815,E2 -11740.815} C_VEL
LIN {X 0,Y 390.038,Z 256.902,A -85,B 0,C 180,E1 -11743.886,E2 -11743.886} C_VEL
LIN {X 0,Y 390.041,Z 256.896,A -85,B 0,C 180,E1 -11746.789,E2 -11746.789} C_VEL
LIN {X 0,Y 390.005,Z 256.906,A -85,B 0,C 180,E1 -11749.556,E2 -11749.556} C_VEL
LIN {X 0,Y 390.033,Z 256.897,A -85,B 0,C 180,E1 -11752.452,E2 -11752.452} C_VEL
LIN {X 0,Y 390.059,Z 256.896,A -85,B 0,C 180,E1 -11756.046,E2 -11756.046} C_VEL
LIN {X 0,Y 390.039,Z 256.899,A -85,B 0,C 180,E1 -11759.872,E2 -11759.872} C_VEL
LIN {X 0,Y 390.025,Z 256.902,A -85,B 0,C 180,E1 -11763.226,E2 -11763.226} C_VEL
LIN {X 0,Y 390.056,Z 256.895,A -85,B 0,C 180,E1 -11766.769,E2 -11766.769} C_VEL
LIN {X 0,Y 390.072,Z 256.893,A -85,B 0,C 180,E1 -11769.982,E2 -11769.982} C_VEL
LIN {X 0,Y 390.105,Z 256.894,A -85,B 0,C 180,E1 -11773.248,E2 -11773.248} C_VEL
LIN {X 0,Y 390.134,Z 256.884,A -85,B 0,C 180,E1 -11776.602,E2 -11776.602} C_VEL
LIN {X 0,Y 390.205,Z 257.098,A -85,B 0,C 180,E1 -11778.31,E2 -11778.31} C_VEL
LIN {X 0,Y 390.465,Z 258.263,A -85,B 0,C 180,E1 -11778.479,E2 -11778.479} C_VEL
LIN {X 0,Y 396.314,Z 274.117,A -85,B 0,C 180,E1 -11779.057,E2 -11779.057} C_VEL
LIN {X 0,Y 395.471,Z 344.52,A -85,B 0,C 180,E1 -11780.35,E2 -11780.35} C_VEL
LIN {X 0,Y 395.334,Z 356.813,A -85,B 0,C 180,E1 -11780.762,E2 -11780.762} C_VEL
LIN {X 0,Y 394.987,Z 367.972,A -85,B 0,C 180,E1 -11781.302,E2 -11781.302} C_VEL
LIN {X 0,Y 394.556,Z 379.686,A -85,B 0,C 180,E1 -11782.066,E2 -11782.066} C_VEL
LIN {X 0,Y 393.953,Z 390.351,A -85,B 0,C 180,E1 -11782.956,E2 -11782.956} C_VEL
LIN {X 0,Y 393.268,Z 401.241,A -85,B 0,C 180,E1 -11784.103,E2 -11784.103} C_VEL
LIN {X 0,Y 392.6,Z 410.935,A -85,B 0,C 180,E1 -11785.38,E2 -11785.38} C_VEL
LIN {X 0,Y 391.83,Z 420.354,A -85,B 0,C 180,E1 -11786.916,E2 -11786.916} C_VEL
LIN {X 0,Y 391.118,Z 427.864,A -85,B 0,C 180,E1 -11788.456,E2 -11788.456} C_VEL
LIN {X 0,Y 390.687,Z 433.881,A -85,B 0,C 180,E1 -11790,E2 -11790} C_VEL
LIN {X 0,Y 390.282,Z 438.676,A -85,B 0,C 180,E1 -11791.548,E2 -11791.548} C_VEL
LIN {X 0,Y 389.918,Z 442.389,A -85,B 0,C 180,E1 -11793.1,E2 -11793.1} C_VEL
LIN {X 0,Y 389.832,Z 444.296,A -85,B 0,C 180,E1 -11794.136,E2 -11794.136} C_VEL
LIN {X 0,Y 389.85,Z 445.786,A -85,B 0,C 180,E1 -11795.172,E2 -11795.172} C_VEL
LIN {X 0,Y 389.75,Z 447.53,A -85,B 0,C 180,E1 -11797.252,E2 -11797.252} C_VEL
LIN {X 0,Y 389.792,Z 447.752,A -85,B 0,C 180,E1 -11799.339,E2 -11799.339} C_VEL
LIN {X 0,Y 389.944,Z 446.343,A -85,B 0,C 180,E1 -11801.435,E2 -11801.435} C_VEL
LIN {X 0,Y 390.353,Z 443.755,A -85,B 0,C 180,E1 -11803.264,E2 -11803.264} C_VEL
LIN {X 0,Y 389.92,Z 442.34,A -85,B 0,C 180,E1 -11804.105,E2 -11804.105} C_VEL
LIN {X 0,Y 387.503,Z 439.732,A -85,B 0,C 180,E1 -11805.471,E2 -11805.471} C_VEL
LIN {X 0,Y 385.146,Z 436.365,A -85,B 0,C 180,E1 -11806.811,E2 -11806.811} C_VEL
LIN {X 0,Y 384.808,Z 433.758,A -85,B 0,C 180,E1 -11807.6,E2 -11807.6} C_VEL
LIN {X 0,Y 385.565,Z 427.543,A -85,B 0,C 180,E1 -11809.154,E2 -11809.154} C_VEL
LIN {X 0,Y 386.537,Z 419.466,A -85,B 0,C 180,E1 -11810.766,E2 -11810.766} C_VEL
LIN {X 0,Y 387.526,Z 410.666,A -85,B 0,C 180,E1 -11812.181,E2 -11812.181} C_VEL
LIN {X 0,Y 388.423,Z 400.833,A -85,B 0,C 180,E1 -11813.457,E2 -11813.457} C_VEL
LIN {X 0,Y 389.273,Z 390.509,A -85,B 0,C 180,E1 -11814.535,E2 -11814.535} C_VEL
LIN {X 0,Y 390.179,Z 379.138,A -85,B 0,C 180,E1 -11815.47,E2 -11815.47} C_VEL
LIN {X 0,Y 390.772,Z 366.882,A -85,B 0,C 180,E1 -11816.245,E2 -11816.245} C_VEL
LIN {X 0,Y 391.099,Z 353.495,A -85,B 0,C 180,E1 -11816.846,E2 -11816.846} C_VEL
LIN {X 0,Y 391.254,Z 340.924,A -85,B 0,C 180,E1 -11817.199,E2 -11817.199} C_VEL
LIN {X 0,Y 392.216,Z 278.771,A -85,B 0,C 180,E1 -11818.356,E2 -11818.356} C_VEL
LIN {X 0,Y 383.298,Z 258.892,A -85,B 0,C 180,E1 -11819.375,E2 -11819.375} C_VEL
LIN {X 0,Y 383.056,Z 257.875,A -85,B 0,C 180,E1 -11819.587,E2 -11819.587} C_VEL
LIN {X 0,Y 383.001,Z 257.78,A -85,B 0,C 180,E1 -11823.401,E2 -11823.401} C_VEL
LIN {X 0,Y 383.023,Z 257.735,A -85,B 0,C 180,E1 -11826.162,E2 -11826.162} C_VEL
LIN {X 0,Y 382.986,Z 257.779,A -85,B 0,C 180,E1 -11829.58,E2 -11829.58} C_VEL
LIN {X 0,Y 383.006,Z 257.769,A -85,B 0,C 180,E1 -11832.778,E2 -11832.778} C_VEL
LIN {X 0,Y 382.988,Z 257.771,A -85,B 0,C 180,E1 -11835.787,E2 -11835.787} C_VEL
LIN {X 0,Y 382.96,Z 257.783,A -85,B 0,C 180,E1 -11838.8,E2 -11838.8} C_VEL
LIN {X 0,Y 382.99,Z 257.759,A -85,B 0,C 180,E1 -11842.097,E2 -11842.097} C_VEL
LIN {X 0,Y 383.015,Z 257.774,A -85,B 0,C 180,E1 -11845.331,E2 -11845.331} C_VEL
LIN {X 0,Y 382.979,Z 257.754,A -85,B 0,C 180,E1 -11849.081,E2 -11849.081} C_VEL
LIN {X 0,Y 382.978,Z 257.78,A -85,B 0,C 180,E1 -11852.692,E2 -11852.692} C_VEL
LIN {X 0,Y 383.009,Z 257.759,A -85,B 0,C 180,E1 -11856.191,E2 -11856.191} C_VEL
LIN {X 0,Y 383.051,Z 257.745,A -85,B 0,C 180,E1 -11859.598,E2 -11859.598} C_VEL
LIN {X 0,Y 383.1,Z 257.762,A -85,B 0,C 180,E1 -11862.931,E2 -11862.931} C_VEL
LIN {X 0,Y 383.121,Z 257.759,A -85,B 0,C 180,E1 -11866.464,E2 -11866.464} C_VEL
LIN {X 0,Y 383.136,Z 257.747,A -85,B 0,C 180,E1 -11870.497,E2 -11870.497} C_VEL
LIN {X 0,Y 383.227,Z 257.751,A -85,B 0,C 180,E1 -11873.682,E2 -11873.682} C_VEL
LIN {X 0,Y 383.365,Z 257.731,A -85,B 0,C 180,E1 -11877.899,E2 -11877.899} C_VEL
LIN {X 0,Y 383.369,Z 257.721,A -85,B 0,C 180,E1 -11882.101,E2 -11882.101} C_VEL
LIN {X 0,Y 383.222,Z 257.742,A -85,B 0,C 180,E1 -11886.317,E2 -11886.317} C_VEL
LIN {X 0,Y 383.136,Z 257.759,A -85,B 0,C 180,E1 -11889.502,E2 -11889.502} C_VEL
LIN {X 0,Y 383.12,Z 257.754,A -85,B 0,C 180,E1 -11893.536,E2 -11893.536} C_VEL
LIN {X 0,Y 383.07,Z 257.764,A -85,B 0,C 180,E1 -11897.445,E2 -11897.445} C_VEL
LIN {X 0,Y 383.023,Z 257.773,A -85,B 0,C 180,E1 -11900.647,E2 -11900.647} C_VEL
LIN {X 0,Y 383.002,Z 257.776,A -85,B 0,C 180,E1 -11903.809,E2 -11903.809} C_VEL
LIN {X 0,Y 382.963,Z 257.762,A -85,B 0,C 180,E1 -11907.309,E2 -11907.309} C_VEL
LIN {X 0,Y 382.974,Z 257.783,A -85,B 0,C 180,E1 -11910.919,E2 -11910.919} C_VEL
LIN {X 0,Y 383.012,Z 257.763,A -85,B 0,C 180,E1 -11914.669,E2 -11914.669} C_VEL
LIN {X 0,Y 382.988,Z 257.772,A -85,B 0,C 180,E1 -11917.902,E2 -11917.902} C_VEL
LIN {X 0,Y 382.956,Z 257.783,A -85,B 0,C 180,E1 -11921.351,E2 -11921.351} C_VEL
LIN {X 0,Y 382.985,Z 257.776,A -85,B 0,C 180,E1 -11924.302,E2 -11924.302} C_VEL
LIN {X 0,Y 382.979,Z 257.777,A -85,B 0,C 180,E1 -11927.236,E2 -11927.236} C_VEL
LIN {X 0,Y 382.982,Z 257.758,A -85,B 0,C 180,E1 -11930.42,E2 -11930.42} C_VEL
LIN {X 0,Y 383.01,Z 257.767,A -85,B 0,C 180,E1 -11934.043,E2 -11934.043} C_VEL
LIN {X 0,Y 383.063,Z 257.938,A -85,B 0,C 180,E1 -11936.606,E2 -11936.606} C_VEL
LIN {X 0,Y 386.272,Z 271.422,A -85,B 0,C 180,E1 -11939.374,E2 -11939.374} C_VEL
LIN {X 0,Y 388.393,Z 281.604,A -85,B 0,C 180,E1 -11941.346,E2 -11941.346} C_VEL
LIN {X 0,Y 387.112,Z 298.123,A -85,B 0,C 180,E1 -11944.169,E2 -11944.169} C_VEL
LIN {X 0,Y 385.486,Z 319.534,A -85,B 0,C 180,E1 -11947.772,E2 -11947.772} C_VEL
LIN {X 0,Y 385.217,Z 323.805,A -85,B 0,C 180,E1 -11948.445,E2 -11948.445} C_VEL
LIN {X 0,Y 388.972,Z 349.625,A -85,B 0,C 180,E1 -11949.214,E2 -11949.214} C_VEL
LIN {X 0,Y 390.916,Z 368.037,A -85,B 0,C 180,E1 -11949.694,E2 -11949.694} C_VEL
LIN {X 0,Y 389.845,Z 434.43,A -85,B 0,C 180,E1 -11950.948,E2 -11950.948} C_VEL
LIN {X 0,Y 389.144,Z 448.025,A -85,B 0,C 180,E1 -11951.405,E2 -11951.405} C_VEL
LIN {X 0,Y 388.19,Z 460.126,A -85,B 0,C 180,E1 -11952.006,E2 -11952.006} C_VEL
LIN {X 0,Y 386.991,Z 472.392,A -85,B 0,C 180,E1 -11952.836,E2 -11952.836} C_VEL
LIN {X 0,Y 385.848,Z 484.036,A -85,B 0,C 180,E1 -11953.873,E2 -11953.873} C_VEL
LIN {X 0,Y 384.724,Z 494.558,A -85,B 0,C 180,E1 -11955.047,E2 -11955.047} C_VEL
LIN {X 0,Y 383.952,Z 503.21,A -85,B 0,C 180,E1 -11956.234,E2 -11956.234} C_VEL
LIN {X 0,Y 383.052,Z 511.213,A -85,B 0,C 180,E1 -11957.55,E2 -11957.55} C_VEL
LIN {X 0,Y 382.419,Z 519.102,A -85,B 0,C 180,E1 -11959.142,E2 -11959.142} C_VEL
LIN {X 0,Y 382.033,Z 526.411,A -85,B 0,C 180,E1 -11961.004,E2 -11961.004} C_VEL
LIN {X 0,Y 381.945,Z 531.331,A -85,B 0,C 180,E1 -11962.599,E2 -11962.599} C_VEL
LIN {X 0,Y 382.041,Z 535.14,A -85,B 0,C 180,E1 -11964.193,E2 -11964.193} C_VEL
LIN {X 0,Y 382.145,Z 537.919,A -85,B 0,C 180,E1 -11965.781,E2 -11965.781} C_VEL
LIN {X 0,Y 382.283,Z 539.252,A -85,B 0,C 180,E1 -11966.838,E2 -11966.838} C_VEL
LIN {X 0,Y 382.216,Z 540.146,A -85,B 0,C 180,E1 -11967.892,E2 -11967.892} C_VEL
LIN {X 0,Y 382.257,Z 540.608,A -85,B 0,C 180,E1 -11968.946,E2 -11968.946} C_VEL
LIN {X 0,Y 382.334,Z 540.675,A -85,B 0,C 180,E1 -11970,E2 -11970} C_VEL
LIN {X 0,Y 382.289,Z 540.33,A -85,B 0,C 180,E1 -11971.053,E2 -11971.053} C_VEL
LIN {X 0,Y 382.264,Z 539.582,A -85,B 0,C 180,E1 -11972.107,E2 -11972.107} C_VEL
LIN {X 0,Y 382.313,Z 538.384,A -85,B 0,C 180,E1 -11973.161,E2 -11973.161} C_VEL
LIN {X 0,Y 382.169,Z 535.77,A -85,B 0,C 180,E1 -11974.746,E2 -11974.746} C_VEL
LIN {X 0,Y 382.067,Z 531.296,A -85,B 0,C 180,E1 -11976.628,E2 -11976.628} C_VEL
LIN {X 0,Y 382.08,Z 525.432,A -85,B 0,C 180,E1 -11978.461,E2 -11978.461} C_VEL
LIN {X 0,Y 382.249,Z 518.888,A -85,B 0,C 180,E1 -11980.059,E2 -11980.059} C_VEL
LIN {X 0,Y 382.693,Z 510.721,A -85,B 0,C 180,E1 -11981.654,E2 -11981.654} C_VEL
LIN {X 0,Y 383.333,Z 502.45,A -85,B 0,C 180,E1 -11982.975,E2 -11982.975} C_VEL
LIN {X 0,Y 383.824,Z 494.696,A -85,B 0,C 180,E1 -11984.013,E2 -11984.013} C_VEL
LIN {X 0,Y 384.624,Z 483.659,A -85,B 0,C 180,E1 -11985.227,E2 -11985.227} C_VEL
LIN {X 0,Y 385.555,Z 473.264,A -85,B 0,C 180,E1 -11986.139,E2 -11986.139} C_VEL
LIN {X 0,Y 386.419,Z 460.856,A -85,B 0,C 180,E1 -11986.985,E2 -11986.985} C_VEL
LIN {X 0,Y 387.305,Z 447.066,A -85,B 0,C 180,E1 -11987.66,E2 -11987.66} C_VEL
LIN {X 0,Y 387.757,Z 433.803,A -85,B 0,C 180,E1 -11988.082,E2 -11988.082} C_VEL
LIN {X 0,Y 388.586,Z 366.607,A -85,B 0,C 180,E1 -11989.327,E2 -11989.327} C_VEL
LIN {X 0,Y 384.229,Z 324.8,A -85,B 0,C 180,E1 -11990.336,E2 -11990.336} C_VEL
LIN {X 0,Y 385.302,Z 304.409,A -85,B 0,C 180,E1 -11993.658,E2 -11993.658} C_VEL
LIN {X 0,Y 386.517,Z 285.746,A -85,B 0,C 180,E1 -11996.744,E2 -11996.744} C_VEL
LIN {X 0,Y 386.969,Z 277.188,A -85,B 0,C 180,E1 -11998.176,E2 -11998.176} C_VEL
LIN {X 0,Y 384.091,Z 262.744,A -85,B 0,C 180,E1 -12000.818,E2 -12000.818} C_VEL
LIN {X 0,Y 383.002,Z 257.895,A -85,B 0,C 180,E1 -12001.762,E2 -12001.762} C_VEL
LIN {X 0,Y 383.006,Z 257.777,A -85,B 0,C 180,E1 -12004.668,E2 -12004.668} C_VEL
LIN {X 0,Y 382.984,Z 257.776,A -85,B 0,C 180,E1 -12007.901,E2 -12007.901} C_VEL
LIN {X 0,Y 382.953,Z 257.785,A -85,B 0,C 180,E1 -12011.35,E2 -12011.35} C_VEL
LIN {X 0,Y 382.981,Z 257.775,A -85,B 0,C 180,E1 -12014.301,E2 -12014.301} C_VEL
LIN {X 0,Y 382.974,Z 257.783,A -85,B 0,C 180,E1 -12017.235,E2 -12017.235} C_VEL
LIN {X 0,Y 382.976,Z 257.776,A -85,B 0,C 180,E1 -12020.418,E2 -12020.418} C_VEL
LIN {X 0,Y 383.003,Z 257.773,A -85,B 0,C 180,E1 -12024.042,E2 -12024.042} C_VEL
LIN {X 0,Y 382.971,Z 257.778,A -85,B 0,C 180,E1 -12027.579,E2 -12027.579} C_VEL
LIN {X 0,Y 382.963,Z 257.778,A -85,B 0,C 180,E1 -12030.298,E2 -12030.298} C_VEL
LIN {X 0,Y 382.992,Z 257.774,A -85,B 0,C 180,E1 -12034.045,E2 -12034.045} C_VEL
LIN {X 0,Y 382.975,Z 257.778,A -85,B 0,C 180,E1 -12037.333,E2 -12037.333} C_VEL
LIN {X 0,Y 383.038,Z 257.774,A -85,B 0,C 180,E1 -12040.715,E2 -12040.715} C_VEL
LIN {X 0,Y 383.064,Z 257.766,A -85,B 0,C 180,E1 -12044.026,E2 -12044.026} C_VEL
LIN {X 0,Y 383.124,Z 257.759,A -85,B 0,C 180,E1 -12047.284,E2 -12047.284} C_VEL
LIN {X 0,Y 383.126,Z 257.762,A -85,B 0,C 180,E1 -12050.497,E2 -12050.497} C_VEL
LIN {X 0,Y 383.216,Z 257.746,A -85,B 0,C 180,E1 -12053.683,E2 -12053.683} C_VEL
LIN {X 0,Y 383.363,Z 257.729,A -85,B 0,C 180,E1 -12057.899,E2 -12057.899} C_VEL
LIN {X 0,Y 383.354,Z 257.732,A -85,B 0,C 180,E1 -12062.102,E2 -12062.102} C_VEL
LIN {X 0,Y 383.199,Z 257.751,A -85,B 0,C 180,E1 -12066.597,E2 -12066.597} C_VEL
LIN {X 0,Y 383.123,Z 257.758,A -85,B 0,C 180,E1 -12069.503,E2 -12069.503} C_VEL
LIN {X 0,Y 383.115,Z 257.759,A -85,B 0,C 180,E1 -12073.537,E2 -12073.537} C_VEL
LIN {X 0,Y 383.065,Z 257.765,A -85,B 0,C 180,E1 -12077.446,E2 -12077.446} C_VEL
LIN {X 0,Y 383.019,Z 257.773,A -85,B 0,C 180,E1 -12080.647,E2 -12080.647} C_VEL
LIN {X 0,Y 382.998,Z 257.777,A -85,B 0,C 180,E1 -12083.81,E2 -12083.81} C_VEL
LIN {X 0,Y 382.959,Z 257.779,A -85,B 0,C 180,E1 -12087.31,E2 -12087.31} C_VEL
LIN {X 0,Y 382.972,Z 257.777,A -85,B 0,C 180,E1 -12090.92,E2 -12090.92} C_VEL
LIN {X 0,Y 383.003,Z 257.773,A -85,B 0,C 180,E1 -12094.67,E2 -12094.67} C_VEL
LIN {X 0,Y 382.984,Z 257.782,A -85,B 0,C 180,E1 -12097.903,E2 -12097.903} C_VEL
LIN {X 0,Y 382.954,Z 257.781,A -85,B 0,C 180,E1 -12101.352,E2 -12101.352} C_VEL
LIN {X 0,Y 382.983,Z 257.777,A -85,B 0,C 180,E1 -12104.303,E2 -12104.303} C_VEL
LIN {X 0,Y 382.977,Z 257.778,A -85,B 0,C 180,E1 -12107.237,E2 -12107.237} C_VEL
LIN {X 0,Y 382.981,Z 257.776,A -85,B 0,C 180,E1 -12110.421,E2 -12110.421} C_VEL
LIN {X 0,Y 383.009,Z 257.774,A -85,B 0,C 180,E1 -12114.044,E2 -12114.044} C_VEL
LIN {X 0,Y 382.979,Z 257.782,A -85,B 0,C 180,E1 -12117.581,E2 -12117.581} C_VEL
LIN {X 0,Y 382.971,Z 257.777,A -85,B 0,C 180,E1 -12120.3,E2 -12120.3} C_VEL
LIN {X 0,Y 383.002,Z 257.774,A -85,B 0,C 180,E1 -12124.046,E2 -12124.046} C_VEL
LIN {X 0,Y 382.985,Z 257.781,A -85,B 0,C 180,E1 -12127.335,E2 -12127.335} C_VEL
LIN {X 0,Y 383.019,Z 257.772,A -85,B 0,C 180,E1 -12130.715,E2 -12130.715} C_VEL
LIN {X 0,Y 383.012,Z 257.772,A -85,B 0,C 180,E1 -12134.025,E2 -12134.025} C_VEL
LIN {X 0,Y 383.112,Z 257.764,A -85,B 0,C 180,E1 -12137.284,E2 -12137.284} C_VEL
LIN {X 0,Y 383.162,Z 257.991,A -85,B 0,C 180,E1 -12137.991,E2 -12137.991} C_VEL
LIN {X 0,Y 383.419,Z 259.064,A -85,B 0,C 180,E1 -12138.153,E2 -12138.153} C_VEL
LIN {X 0,Y 389.514,Z 275.539,A -85,B 0,C 180,E1 -12138.773,E2 -12138.773} C_VEL
LIN {X 0,Y 388.666,Z 345.289,A -85,B 0,C 180,E1 -12140.076,E2 -12140.076} C_VEL
LIN {X 0,Y 388.498,Z 358.443,A -85,B 0,C 180,E1 -12140.532,E2 -12140.532} C_VEL
LIN {X 0,Y 388.135,Z 369.403,A -85,B 0,C 180,E1 -12141.081,E2 -12141.081} C_VEL
LIN {X 0,Y 387.633,Z 381.86,A -85,B 0,C 180,E1 -12141.923,E2 -12141.923} C_VEL
LIN {X 0,Y 386.947,Z 393.524,A -85,B 0,C 180,E1 -12142.959,E2 -12142.959} C_VEL
LIN {X 0,Y 386.199,Z 403.945,A -85,B 0,C 180,E1 -12144.125,E2 -12144.125} C_VEL
LIN {X 0,Y 385.468,Z 414.17,A -85,B 0,C 180,E1 -12145.556,E2 -12145.556} C_VEL
LIN {X 0,Y 384.687,Z 423.053,A -85,B 0,C 180,E1 -12147.121,E2 -12147.121} C_VEL
LIN {X 0,Y 383.985,Z 430.229,A -85,B 0,C 180,E1 -12148.69,E2 -12148.69} C_VEL
LIN {X 0,Y 383.478,Z 436.784,A -85,B 0,C 180,E1 -12150.525,E2 -12150.525} C_VEL
LIN {X 0,Y 383.127,Z 441.126,A -85,B 0,C 180,E1 -12152.103,E2 -12152.103} C_VEL
LIN {X 0,Y 382.864,Z 443.439,A -85,B 0,C 180,E1 -12153.157,E2 -12153.157} C_VEL
LIN {X 0,Y 382.787,Z 445.314,A -85,B 0,C 180,E1 -12154.212,E2 -12154.212} C_VEL
LIN {X 0,Y 382.79,Z 446.75,A -85,B 0,C 180,E1 -12155.267,E2 -12155.267} C_VEL
LIN {X 0,Y 382.691,Z 448.429,A -85,B 0,C 180,E1 -12157.386,E2 -12157.386} C_VEL
LIN {X 0,Y 382.705,Z 448.703,A -85,B 0,C 180,E1 -12158.448,E2 -12158.448} C_VEL
LIN {X 0,Y 382.754,Z 448.564,A -85,B 0,C 180,E1 -12159.512,E2 -12159.512} C_VEL
LIN {X 0,Y 382.946,Z 447.09,A -85,B 0,C 180,E1 -12161.647,E2 -12161.647} C_VEL
LIN {X 0,Y 383.359,Z 444.71,A -85,B 0,C 180,E1 -12163.34,E2 -12163.34} C_VEL
LIN {X 0,Y 383.753,Z 441.728,A -85,B 0,C 180,E1 -12164.856,E2 -12164.856} C_VEL
LIN {X 0,Y 384.306,Z 437.468,A -85,B 0,C 180,E1 -12166.467,E2 -12166.467} C_VEL
LIN {X 0,Y 384.808,Z 433.758,A -85,B 0,C 180,E1 -12167.6,E2 -12167.6} C_VEL
LIN {X 0,Y 384.506,Z 431.008,A -85,B 0,C 180,E1 -12168.374,E2 -12168.374} C_VEL
LIN {X 0,Y 382.355,Z 426.313,A -85,B 0,C 180,E1 -12169.645,E2 -12169.645} C_VEL
LIN {X 0,Y 380.291,Z 421.074,A -85,B 0,C 180,E1 -12170.871,E2 -12170.871} C_VEL
LIN {X 0,Y 380.114,Z 417.363,A -85,B 0,C 180,E1 -12171.563,E2 -12171.563} C_VEL
LIN {X 0,Y 381.041,Z 409.374,A -85,B 0,C 180,E1 -12172.788,E2 -12172.788} C_VEL
LIN {X 0,Y 381.948,Z 399.614,A -85,B 0,C 180,E1 -12174.023,E2 -12174.023} C_VEL
LIN {X 0,Y 382.848,Z 388.817,A -85,B 0,C 180,E1 -12175.119,E2 -12175.119} C_VEL
LIN {X 0,Y 383.626,Z 377.992,A -85,B 0,C 180,E1 -12175.98,E2 -12175.98} C_VEL
LIN {X 0,Y 384.319,Z 364.968,A -85,B 0,C 180,E1 -12176.763,E2 -12176.763} C_VEL
LIN {X 0,Y 384.587,Z 352.733,A -85,B 0,C 180,E1 -12177.291,E2 -12177.291} C_VEL
LIN {X 0,Y 384.715,Z 338.464,A -85,B 0,C 180,E1 -12177.656,E2 -12177.656} C_VEL
LIN {X 0,Y 385.645,Z 280.455,A -85,B 0,C 180,E1 -12178.756,E2 -12178.756} C_VEL
LIN {X 0,Y 376.804,Z 261.206,A -85,B 0,C 180,E1 -12179.769,E2 -12179.769} C_VEL
LIN {X 0,Y 376.058,Z 259.196,A -85,B 0,C 180,E1 -12179.935,E2 -12179.935} C_VEL
LIN {X 0,Y 375.986,Z 258.695,A -85,B 0,C 180,E1 -12180.14,E2 -12180.14} C_VEL
LIN {X 0,Y 375.959,Z 258.65,A -85,B 0,C 180,E1 -12184.111,E2 -12184.111} C_VEL
LIN {X 0,Y 375.949,Z 258.614,A -85,B 0,C 180,E1 -12186.741,E2 -12186.741} C_VEL
LIN {X 0,Y 375.938,Z 258.658,A -85,B 0,C 180,E1 -12189.961,E2 -12189.961} C_VEL
LIN {X 0,Y 375.924,Z 258.659,A -85,B 0,C 180,E1 -12193.766,E2 -12193.766} C_VEL
LIN {X 0,Y 375.931,Z 258.642,A -85,B 0,C 180,E1 -12196.81,E2 -12196.81} C_VEL
LIN {X 0,Y 375.932,Z 258.652,A -85,B 0,C 180,E1 -12200.533,E2 -12200.533} C_VEL
LIN {X 0,Y 375.959,Z 258.639,A -85,B 0,C 180,E1 -12203.495,E2 -12203.495} C_VEL
LIN {X 0,Y 375.958,Z 258.656,A -85,B 0,C 180,E1 -12205.888,E2 -12205.888} C_VEL
LIN {X 0,Y 375.959,Z 258.625,A -85,B 0,C 180,E1 -12209.686,E2 -12209.686} C_VEL
LIN {X 0,Y 375.922,Z 258.652,A -85,B 0,C 180,E1 -12212.135,E2 -12212.135} C_VEL
LIN {X 0,Y 375.957,Z 258.644,A -85,B 0,C 180,E1 -12215.716,E2 -12215.716} C_VEL
LIN {X 0,Y 375.976,Z 258.623,A -85,B 0,C 180,E1 -12219.196,E2 -12219.196} C_VEL
LIN {X 0,Y 376.046,Z 258.642,A -85,B 0,C 180,E1 -12222.6,E2 -12222.6} C_VEL
LIN {X 0,Y 376.085,Z 258.634,A -85,B 0,C 180,E1 -12226.342,E2 -12226.342} C_VEL
LIN {X 0,Y 376.106,Z 258.623,A -85,B 0,C 180,E1 -12230.318,E2 -12230.318} C_VEL
LIN {X 0,Y 376.186,Z 258.627,A -85,B 0,C 180,E1 -12233.564,E2 -12233.564} C_VEL
LIN {X 0,Y 376.33,Z 258.606,A -85,B 0,C 180,E1 -12237.859,E2 -12237.859} C_VEL
LIN {X 0,Y 376.334,Z 258.597,A -85,B 0,C 180,E1 -12242.14,E2 -12242.14} C_VEL
LIN {X 0,Y 376.183,Z 258.618,A -85,B 0,C 180,E1 -12246.436,E2 -12246.436} C_VEL
LIN {X 0,Y 376.106,Z 258.637,A -85,B 0,C 180,E1 -12249.682,E2 -12249.682} C_VEL
LIN {X 0,Y 376.084,Z 258.63,A -85,B 0,C 180,E1 -12253.657,E2 -12253.657} C_VEL
LIN {X 0,Y 376.027,Z 258.641,A -85,B 0,C 180,E1 -12257.4,E2 -12257.4} C_VEL
LIN {X 0,Y 375.974,Z 258.653,A -85,B 0,C 180,E1 -12260.832,E2 -12260.832} C_VEL
LIN {X 0,Y 375.962,Z 258.652,A -85,B 0,C 180,E1 -12264.284,E2 -12264.284} C_VEL
LIN {X 0,Y 375.911,Z 258.64,A -85,B 0,C 180,E1 -12267.865,E2 -12267.865} C_VEL
LIN {X 0,Y 375.932,Z 258.657,A -85,B 0,C 180,E1 -12270.689,E2 -12270.689} C_VEL
LIN {X 0,Y 375.954,Z 258.639,A -85,B 0,C 180,E1 -12274.112,E2 -12274.112} C_VEL
LIN {X 0,Y 375.946,Z 258.658,A -85,B 0,C 180,E1 -12276.742,E2 -12276.742} C_VEL
LIN {X 0,Y 375.934,Z 258.654,A -85,B 0,C 180,E1 -12279.962,E2 -12279.962} C_VEL
LIN {X 0,Y 375.921,Z 258.654,A -85,B 0,C 180,E1 -12283.767,E2 -12283.767} C_VEL
LIN {X 0,Y 375.929,Z 258.653,A -85,B 0,C 180,E1 -12286.811,E2 -12286.811} C_VEL
LIN {X 0,Y 375.93,Z 258.635,A -85,B 0,C 180,E1 -12290.534,E2 -12290.534} C_VEL
LIN {X 0,Y 375.955,Z 258.655,A -85,B 0,C 180,E1 -12293.498,E2 -12293.498} C_VEL
LIN {X 0,Y 376.008,Z 258.863,A -85,B 0,C 180,E1 -12296.195,E2 -12296.195} C_VEL
LIN {X 0,Y 379.349,Z 272.507,A -85,B 0,C 180,E1 -12299.062,E2 -12299.062} C_VEL
LIN {X 0,Y 381.491,Z 282.728,A -85,B 0,C 180,E1 -12301.087,E2 -12301.087} C_VEL
LIN {X 0,Y 381.096,Z 289.465,A -85,B 0,C 180,E1 -12302.276,E2 -12302.276} C_VEL
LIN {X 0,Y 379.278,Z 310.726,A -85,B 0,C 180,E1 -12305.942,E2 -12305.942} C_VEL
LIN {X 0,Y 378.395,Z 322.811,A -85,B 0,C 180,E1 -12307.976,E2 -12307.976} C_VEL
LIN {X 0,Y 382.154,Z 348.266,A -85,B 0,C 180,E1 -12308.758,E2 -12308.758} C_VEL
LIN {X 0,Y 384.339,Z 368.419,A -85,B 0,C 180,E1 -12309.301,E2 -12309.301} C_VEL
LIN {X 0,Y 383.206,Z 434.218,A -85,B 0,C 180,E1 -12310.572,E2 -12310.572} C_VEL
LIN {X 0,Y 382.49,Z 447.533,A -85,B 0,C 180,E1 -12311.035,E2 -12311.035} C_VEL
LIN {X 0,Y 381.441,Z 460.1,A -85,B 0,C 180,E1 -12311.677,E2 -12311.677} C_VEL
LIN {X 0,Y 380.204,Z 472.115,A -85,B 0,C 180,E1 -12312.52,E2 -12312.52} C_VEL
LIN {X 0,Y 379.017,Z 483.65,A -85,B 0,C 180,E1 -12313.574,E2 -12313.574} C_VEL
LIN {X 0,Y 377.799,Z 494.083,A -85,B 0,C 180,E1 -12314.766,E2 -12314.766} C_VEL
LIN {X 0,Y 377.02,Z 502.67,A -85,B 0,C 180,E1 -12315.976,E2 -12315.976} C_VEL
LIN {X 0,Y 375.958,Z 512.013,A -85,B 0,C 180,E1 -12317.586,E2 -12317.586} C_VEL
LIN {X 0,Y 375.286,Z 519.578,A -85,B 0,C 180,E1 -12319.206,E2 -12319.206} C_VEL
LIN {X 0,Y 374.954,Z 525.706,A -85,B 0,C 180,E1 -12320.832,E2 -12320.832} C_VEL
LIN {X 0,Y 374.866,Z 530.594,A -85,B 0,C 180,E1 -12322.459,E2 -12322.459} C_VEL
LIN {X 0,Y 374.963,Z 534.373,A -85,B 0,C 180,E1 -12324.083,E2 -12324.083} C_VEL
LIN {X 0,Y 375.068,Z 537.125,A -85,B 0,C 180,E1 -12325.701,E2 -12325.701} C_VEL
LIN {X 0,Y 375.215,Z 538.446,A -85,B 0,C 180,E1 -12326.778,E2 -12326.778} C_VEL
LIN {X 0,Y 375.165,Z 539.318,A -85,B 0,C 180,E1 -12327.852,E2 -12327.852} C_VEL
LIN {X 0,Y 375.204,Z 539.764,A -85,B 0,C 180,E1 -12328.926,E2 -12328.926} C_VEL
LIN {X 0,Y 375.285,Z 539.819,A -85,B 0,C 180,E1 -12330,E2 -12330} C_VEL
LIN {X 0,Y 375.238,Z 539.46,A -85,B 0,C 180,E1 -12331.073,E2 -12331.073} C_VEL
LIN {X 0,Y 375.214,Z 538.689,A -85,B 0,C 180,E1 -12332.146,E2 -12332.146} C_VEL
LIN {X 0,Y 375.267,Z 537.472,A -85,B 0,C 180,E1 -12333.22,E2 -12333.22} C_VEL
LIN {X 0,Y 375.096,Z 534.823,A -85,B 0,C 180,E1 -12334.836,E2 -12334.836} C_VEL
LIN {X 0,Y 375.003,Z 530.615,A -85,B 0,C 180,E1 -12336.644,E2 -12336.644} C_VEL
LIN {X 0,Y 375.008,Z 524.411,A -85,B 0,C 180,E1 -12338.622,E2 -12338.622} C_VEL
LIN {X 0,Y 375.188,Z 517.807,A -85,B 0,C 180,E1 -12340.25,E2 -12340.25} C_VEL
LIN {X 0,Y 375.673,Z 509.593,A -85,B 0,C 180,E1 -12341.875,E2 -12341.875} C_VEL
LIN {X 0,Y 376.385,Z 499.902,A -85,B 0,C 180,E1 -12343.423,E2 -12343.423} C_VEL
LIN {X 0,Y 377.172,Z 489.867,A -85,B 0,C 180,E1 -12344.706,E2 -12344.706} C_VEL
LIN {X 0,Y 377.986,Z 479.523,A -85,B 0,C 180,E1 -12345.778,E2 -12345.778} C_VEL
LIN {X 0,Y 378.917,Z 468.258,A -85,B 0,C 180,E1 -12346.707,E2 -12346.707} C_VEL
LIN {X 0,Y 379.876,Z 455.72,A -85,B 0,C 180,E1 -12347.495,E2 -12347.495} C_VEL
LIN {X 0,Y 380.609,Z 442.315,A -85,B 0,C 180,E1 -12348.085,E2 -12348.085} C_VEL
LIN {X 0,Y 380.97,Z 429.585,A -85,B 0,C 180,E1 -12348.441,E2 -12348.441} C_VEL
LIN {X 0,Y 381.652,Z 366.496,A -85,B 0,C 180,E1 -12349.623,E2 -12349.623} C_VEL
LIN {X 0,Y 377.235,Z 323.985,A -85,B 0,C 180,E1 -12350.666,E2 -12350.666} C_VEL
LIN {X 0,Y 378.208,Z 306.583,A -85,B 0,C 180,E1 -12353.547,E2 -12353.547} C_VEL
LIN {X 0,Y 379.509,Z 288.121,A -85,B 0,C 180,E1 -12356.653,E2 -12356.653} C_VEL
LIN {X 0,Y 380.058,Z 279.409,A -85,B 0,C 180,E1 -12358.133,E2 -12358.133} C_VEL
LIN {X 0,Y 378.394,Z 269.932,A -85,B 0,C 180,E1 -12359.876,E2 -12359.876} C_VEL
LIN {X 0,Y 375.996,Z 258.773,A -85,B 0,C 180,E1 -12362.03,E2 -12362.03} C_VEL
LIN {X 0,Y 375.943,Z 258.659,A -85,B 0,C 180,E1 -12365.416,E2 -12365.416} C_VEL
LIN {X 0,Y 375.926,Z 258.654,A -85,B 0,C 180,E1 -12368.261,E2 -12368.261} C_VEL
LIN {X 0,Y 375.906,Z 258.66,A -85,B 0,C 180,E1 -12371.596,E2 -12371.596} C_VEL
LIN {X 0,Y 375.913,Z 258.658,A -85,B 0,C 180,E1 -12374.729,E2 -12374.729} C_VEL
LIN {X 0,Y 375.899,Z 258.659,A -85,B 0,C 180,E1 -12377.695,E2 -12377.695} C_VEL
LIN {X 0,Y 375.925,Z 258.655,A -85,B 0,C 180,E1 -12380.533,E2 -12380.533} C_VEL
LIN {X 0,Y 375.948,Z 258.654,A -85,B 0,C 180,E1 -12383.496,E2 -12383.496} C_VEL
LIN {X 0,Y 375.948,Z 258.652,A -85,B 0,C 180,E1 -12385.887,E2 -12385.887} C_VEL
LIN {X 0,Y 375.95,Z 258.652,A -85,B 0,C 180,E1 -12389.686,E2 -12389.686} C_VEL
LIN {X 0,Y 375.905,Z 258.657,A -85,B 0,C 180,E1 -12392.134,E2 -12392.134} C_VEL
LIN {X 0,Y 375.956,Z 258.651,A -85,B 0,C 180,E1 -12395.716,E2 -12395.716} C_VEL
LIN {X 0,Y 375.949,Z 258.654,A -85,B 0,C 180,E1 -12399.195,E2 -12399.195} C_VEL
LIN {X 0,Y 376.021,Z 258.647,A -85,B 0,C 180,E1 -12402.6,E2 -12402.6} C_VEL
LIN {X 0,Y 376.079,Z 258.638,A -85,B 0,C 180,E1 -12406.342,E2 -12406.342} C_VEL
LIN {X 0,Y 376.097,Z 258.636,A -85,B 0,C 180,E1 -12410.318,E2 -12410.318} C_VEL
LIN {X 0,Y 376.177,Z 258.623,A -85,B 0,C 180,E1 -12413.564,E2 -12413.564} C_VEL
LIN {X 0,Y 376.328,Z 258.605,A -85,B 0,C 180,E1 -12417.86,E2 -12417.86} C_VEL
LIN {X 0,Y 376.318,Z 258.608,A -85,B 0,C 180,E1 -12422.141,E2 -12422.141} C_VEL
LIN {X 0,Y 376.167,Z 258.629,A -85,B 0,C 180,E1 -12426.584,E2 -12426.584} C_VEL
LIN {X 0,Y 376.094,Z 258.634,A -85,B 0,C 180,E1 -12429.682,E2 -12429.682} C_VEL
LIN {X 0,Y 376.079,Z 258.636,A -85,B 0,C 180,E1 -12433.658,E2 -12433.658} C_VEL
LIN {X 0,Y 376.017,Z 258.644,A -85,B 0,C 180,E1 -12437.6,E2 -12437.6} C_VEL
LIN {X 0,Y 375.969,Z 258.65,A -85,B 0,C 180,E1 -12440.833,E2 -12440.833} C_VEL
LIN {X 0,Y 375.948,Z 258.656,A -85,B 0,C 180,E1 -12444.285,E2 -12444.285} C_VEL
LIN {X 0,Y 375.908,Z 258.661,A -85,B 0,C 180,E1 -12447.866,E2 -12447.866} C_VEL
LIN {X 0,Y 375.947,Z 258.654,A -85,B 0,C 180,E1 -12451.563,E2 -12451.563} C_VEL
LIN {X 0,Y 375.941,Z 258.654,A -85,B 0,C 180,E1 -12455.418,E2 -12455.418} C_VEL
LIN {X 0,Y 375.926,Z 258.657,A -85,B 0,C 180,E1 -12458.264,E2 -12458.264} C_VEL
LIN {X 0,Y 375.907,Z 258.661,A -85,B 0,C 180,E1 -12461.598,E2 -12461.598} C_VEL
LIN {X 0,Y 375.914,Z 258.656,A -85,B 0,C 180,E1 -12464.731,E2 -12464.731} C_VEL
LIN {X 0,Y 375.902,Z 258.664,A -85,B 0,C 180,E1 -12467.697,E2 -12467.697} C_VEL
LIN {X 0,Y 375.929,Z 258.654,A -85,B 0,C 180,E1 -12470.535,E2 -12470.535} C_VEL
LIN {X 0,Y 375.953,Z 258.656,A -85,B 0,C 180,E1 -12473.499,E2 -12473.499} C_VEL
LIN {X 0,Y 375.955,Z 258.654,A -85,B 0,C 180,E1 -12475.889,E2 -12475.889} C_VEL
LIN {X 0,Y 375.958,Z 258.655,A -85,B 0,C 180,E1 -12479.688,E2 -12479.688} C_VEL
LIN {X 0,Y 375.915,Z 258.657,A -85,B 0,C 180,E1 -12482.136,E2 -12482.136} C_VEL
LIN {X 0,Y 375.934,Z 258.653,A -85,B 0,C 180,E1 -12484.535,E2 -12484.535} C_VEL
LIN {X 0,Y 375.968,Z 258.651,A -85,B 0,C 180,E1 -12486.888,E2 -12486.888} C_VEL
LIN {X 0,Y 375.964,Z 258.65,A -85,B 0,C 180,E1 -12490.338,E2 -12490.338} C_VEL
LIN {X 0,Y 375.97,Z 258.651,A -85,B 0,C 180,E1 -12493.717,E2 -12493.717} C_VEL
LIN {X 0,Y 376.077,Z 258.726,A -85,B 0,C 180,E1 -12497.591,E2 -12497.591} C_VEL
LIN {X 0,Y 376.22,Z 259.483,A -85,B 0,C 180,E1 -12497.783,E2 -12497.783} C_VEL
LIN {X 0,Y 382.624,Z 276.706,A -85,B 0,C 180,E1 -12498.47,E2 -12498.47} C_VEL
LIN {X 0,Y 381.837,Z 346.196,A -85,B 0,C 180,E1 -12499.797,E2 -12499.797} C_VEL
LIN {X 0,Y 381.677,Z 359.317,A -85,B 0,C 180,E1 -12500.261,E2 -12500.261} C_VEL
LIN {X 0,Y 381.326,Z 370.806,A -85,B 0,C 180,E1 -12500.854,E2 -12500.854} C_VEL
LIN {X 0,Y 380.799,Z 382.288,A -85,B 0,C 180,E1 -12501.644,E2 -12501.644} C_VEL
LIN {X 0,Y 380.143,Z 392.778,A -85,B 0,C 180,E1 -12502.565,E2 -12502.565} C_VEL
LIN {X 0,Y 379.389,Z 403.489,A -85,B 0,C 180,E1 -12503.753,E2 -12503.753} C_VEL
LIN {X 0,Y 378.628,Z 413.959,A -85,B 0,C 180,E1 -12505.209,E2 -12505.209} C_VEL
LIN {X 0,Y 377.96,Z 421.7,A -85,B 0,C 180,E1 -12506.536,E2 -12506.536} C_VEL
LIN {X 0,Y 377.184,Z 429.293,A -85,B 0,C 180,E1 -12508.132,E2 -12508.132} C_VEL
LIN {X 0,Y 376.716,Z 434.475,A -85,B 0,C 180,E1 -12509.466,E2 -12509.466} C_VEL
LIN {X 0,Y 376.271,Z 439.508,A -85,B 0,C 180,E1 -12511.071,E2 -12511.071} C_VEL
LIN {X 0,Y 375.932,Z 443.427,A -85,B 0,C 180,E1 -12512.679,E2 -12512.679} C_VEL
LIN {X 0,Y 375.743,Z 446.325,A -85,B 0,C 180,E1 -12514.291,E2 -12514.291} C_VEL
LIN {X 0,Y 375.732,Z 447.705,A -85,B 0,C 180,E1 -12515.367,E2 -12515.367} C_VEL
LIN {X 0,Y 375.653,Z 449.325,A -85,B 0,C 180,E1 -12517.525,E2 -12517.525} C_VEL
LIN {X 0,Y 375.673,Z 449.563,A -85,B 0,C 180,E1 -12518.608,E2 -12518.608} C_VEL
LIN {X 0,Y 375.804,Z 448.799,A -85,B 0,C 180,E1 -12520.779,E2 -12520.779} C_VEL
LIN {X 0,Y 375.954,Z 447.839,A -85,B 0,C 180,E1 -12521.867,E2 -12521.867} C_VEL
LIN {X 0,Y 376.479,Z 444.898,A -85,B 0,C 180,E1 -12523.897,E2 -12523.897} C_VEL
LIN {X 0,Y 376.993,Z 441.031,A -85,B 0,C 180,E1 -12525.683,E2 -12525.683} C_VEL
LIN {X 0,Y 377.645,Z 436.3,A -85,B 0,C 180,E1 -12527.323,E2 -12527.323} C_VEL
LIN {X 0,Y 378.43,Z 430.489,A -85,B 0,C 180,E1 -12528.911,E2 -12528.911} C_VEL
LIN {X 0,Y 379.462,Z 422.716,A -85,B 0,C 180,E1 -12530.603,E2 -12530.603} C_VEL
LIN {X 0,Y 380.114,Z 417.363,A -85,B 0,C 180,E1 -12531.563,E2 -12531.563} C_VEL
LIN {X 0,Y 379.957,Z 413.485,A -85,B 0,C 180,E1 -12532.231,E2 -12532.231} C_VEL
LIN {X 0,Y 378.005,Z 407.033,A -85,B 0,C 180,E1 -12533.329,E2 -12533.329} C_VEL
LIN {X 0,Y 376.01,Z 400.121,A -85,B 0,C 180,E1 -12534.361,E2 -12534.361} C_VEL
LIN {X 0,Y 375.773,Z 395.454,A -85,B 0,C 180,E1 -12534.914,E2 -12534.914} C_VEL
LIN {X 0,Y 376.608,Z 385.709,A -85,B 0,C 180,E1 -12535.823,E2 -12535.823} C_VEL
LIN {X 0,Y 377.361,Z 374.414,A -85,B 0,C 180,E1 -12536.658,E2 -12536.658} C_VEL
LIN {X 0,Y 377.899,Z 361.283,A -85,B 0,C 180,E1 -12537.376,E2 -12537.376} C_VEL
LIN {X 0,Y 378.143,Z 348.534,A -85,B 0,C 180,E1 -12537.849,E2 -12537.849} C_VEL
LIN {X 0,Y 378.624,Z 311.68,A -85,B 0,C 180,E1 -12538.598,E2 -12538.598} C_VEL
LIN {X 0,Y 379.243,Z 282.485,A -85,B 0,C 180,E1 -12539.154,E2 -12539.154} C_VEL
LIN {X 0,Y 370.111,Z 262.662,A -85,B 0,C 180,E1 -12540.232,E2 -12540.232} C_VEL
LIN {X 0,Y 369.078,Z 260.294,A -85,B 0,C 180,E1 -12540.401,E2 -12540.401} C_VEL
LIN {X 0,Y 368.909,Z 259.573,A -85,B 0,C 180,E1 -12540.655,E2 -12540.655} C_VEL
LIN {X 0,Y 368.897,Z 259.537,A -85,B 0,C 180,E1 -12543.538,E2 -12543.538} C_VEL
LIN {X 0,Y 368.896,Z 259.492,A -85,B 0,C 180,E1 -12546.854,E2 -12546.854} C_VEL
LIN {X 0,Y 368.884,Z 259.538,A -85,B 0,C 180,E1 -12550.373,E2 -12550.373} C_VEL
LIN {X 0,Y 368.878,Z 259.536,A -85,B 0,C 180,E1 -12553.614,E2 -12553.614} C_VEL
LIN {X 0,Y 368.881,Z 259.519,A -85,B 0,C 180,E1 -12556.695,E2 -12556.695} C_VEL
LIN {X 0,Y 368.883,Z 259.535,A -85,B 0,C 180,E1 -12559.648,E2 -12559.648} C_VEL
LIN {X 0,Y 368.896,Z 259.515,A -85,B 0,C 180,E1 -12563.145,E2 -12563.145} C_VEL
LIN {X 0,Y 368.894,Z 259.534,A -85,B 0,C 180,E1 -12566.461,E2 -12566.461} C_VEL
LIN {X 0,Y 368.91,Z 259.505,A -85,B 0,C 180,E1 -12569.044,E2 -12569.044} C_VEL
LIN {X 0,Y 368.907,Z 259.521,A -85,B 0,C 180,E1 -12571.557,E2 -12571.557} C_VEL
LIN {X 0,Y 368.912,Z 259.527,A -85,B 0,C 180,E1 -12575.221,E2 -12575.221} C_VEL
LIN {X 0,Y 368.906,Z 259.498,A -85,B 0,C 180,E1 -12578.779,E2 -12578.779} C_VEL
LIN {X 0,Y 368.987,Z 259.524,A -85,B 0,C 180,E1 -12582.257,E2 -12582.257} C_VEL
LIN {X 0,Y 369.033,Z 259.511,A -85,B 0,C 180,E1 -12586.228,E2 -12586.228} C_VEL
LIN {X 0,Y 369.056,Z 259.502,A -85,B 0,C 180,E1 -12590.131,E2 -12590.131} C_VEL
LIN {X 0,Y 369.148,Z 259.502,A -85,B 0,C 180,E1 -12593.44,E2 -12593.44} C_VEL
LIN {X 0,Y 369.294,Z 259.482,A -85,B 0,C 180,E1 -12597.818,E2 -12597.818} C_VEL
LIN {X 0,Y 369.298,Z 259.473,A -85,B 0,C 180,E1 -12602.181,E2 -12602.181} C_VEL
LIN {X 0,Y 369.145,Z 259.495,A -85,B 0,C 180,E1 -12606.559,E2 -12606.559} C_VEL
LIN {X 0,Y 369.056,Z 259.514,A -85,B 0,C 180,E1 -12609.868,E2 -12609.868} C_VEL
LIN {X 0,Y 369.032,Z 259.509,A -85,B 0,C 180,E1 -12613.772,E2 -12613.772} C_VEL
LIN {X 0,Y 368.986,Z 259.516,A -85,B 0,C 180,E1 -12617.743,E2 -12617.743} C_VEL
LIN {X 0,Y 368.904,Z 259.531,A -85,B 0,C 180,E1 -12621.221,E2 -12621.221} C_VEL
LIN {X 0,Y 368.917,Z 259.532,A -85,B 0,C 180,E1 -12624.778,E2 -12624.778} C_VEL
LIN {X 0,Y 368.887,Z 259.521,A -85,B 0,C 180,E1 -12628.792,E2 -12628.792} C_VEL
LIN {X 0,Y 368.885,Z 259.531,A -85,B 0,C 180,E1 -12632.239,E2 -12632.239} C_VEL
LIN {X 0,Y 368.923,Z 259.521,A -85,B 0,C 180,E1 -12635.001,E2 -12635.001} C_VEL
LIN {X 0,Y 368.872,Z 259.527,A -85,B 0,C 180,E1 -12638.634,E2 -12638.634} C_VEL
LIN {X 0,Y 368.855,Z 259.538,A -85,B 0,C 180,E1 -12642.006,E2 -12642.006} C_VEL
LIN {X 0,Y 368.87,Z 259.537,A -85,B 0,C 180,E1 -12645.175,E2 -12645.175} C_VEL
LIN {X 0,Y 368.857,Z 259.54,A -85,B 0,C 180,E1 -12648.175,E2 -12648.175} C_VEL
LIN {X 0,Y 368.873,Z 259.516,A -85,B 0,C 180,E1 -12651.367,E2 -12651.367} C_VEL
LIN {X 0,Y 368.929,Z 259.514,A -85,B 0,C 180,E1 -12655.146,E2 -12655.146} C_VEL
LIN {X 0,Y 368.967,Z 259.808,A -85,B 0,C 180,E1 -12655.771,E2 -12655.771} C_VEL
LIN {X 0,Y 372.469,Z 273.888,A -85,B 0,C 180,E1 -12658.798,E2 -12658.798} C_VEL
LIN {X 0,Y 374.563,Z 283.773,A -85,B 0,C 180,E1 -12660.801,E2 -12660.801} C_VEL
LIN {X 0,Y 374.578,Z 287.432,A -85,B 0,C 180,E1 -12661.478,E2 -12661.478} C_VEL
LIN {X 0,Y 372.811,Z 306.317,A -85,B 0,C 180,E1 -12664.805,E2 -12664.805} C_VEL
LIN {X 0,Y 371.617,Z 321.943,A -85,B 0,C 180,E1 -12667.493,E2 -12667.493} C_VEL
LIN {X 0,Y 375.618,Z 349.009,A -85,B 0,C 180,E1 -12668.346,E2 -12668.346} C_VEL
LIN {X 0,Y 377.748,Z 368.784,A -85,B 0,C 180,E1 -12668.891,E2 -12668.891} C_VEL
LIN {X 0,Y 376.633,Z 432.975,A -85,B 0,C 180,E1 -12670.153,E2 -12670.153} C_VEL
LIN {X 0,Y 375.925,Z 446.311,A -85,B 0,C 180,E1 -12670.62,E2 -12670.62} C_VEL
LIN {X 0,Y 374.86,Z 458.969,A -85,B 0,C 180,E1 -12671.273,E2 -12671.273} C_VEL
LIN {X 0,Y 373.617,Z 470.263,A -85,B 0,C 180,E1 -12672.06,E2 -12672.06} C_VEL
LIN {X 0,Y 372.352,Z 481.974,A -85,B 0,C 180,E1 -12673.13,E2 -12673.13} C_VEL
LIN {X 0,Y 371.02,Z 492.539,A -85,B 0,C 180,E1 -12674.34,E2 -12674.34} C_VEL
LIN {X 0,Y 370.019,Z 502.125,A -85,B 0,C 180,E1 -12675.705,E2 -12675.705} C_VEL
LIN {X 0,Y 369.119,Z 510.013,A -85,B 0,C 180,E1 -12677.072,E2 -12677.072} C_VEL
LIN {X 0,Y 368.399,Z 517.779,A -85,B 0,C 180,E1 -12678.723,E2 -12678.723} C_VEL
LIN {X 0,Y 367.896,Z 525.007,A -85,B 0,C 180,E1 -12680.655,E2 -12680.655} C_VEL
LIN {X 0,Y 367.776,Z 529.859,A -85,B 0,C 180,E1 -12682.312,E2 -12682.312} C_VEL
LIN {X 0,Y 367.889,Z 533.217,A -85,B 0,C 180,E1 -12683.775,E2 -12683.775} C_VEL
LIN {X 0,Y 367.979,Z 536.331,A -85,B 0,C 180,E1 -12685.618,E2 -12685.618} C_VEL
LIN {X 0,Y 368.133,Z 537.64,A -85,B 0,C 180,E1 -12686.716,E2 -12686.716} C_VEL
LIN {X 0,Y 368.114,Z 538.488,A -85,B 0,C 180,E1 -12687.811,E2 -12687.811} C_VEL
LIN {X 0,Y 368.236,Z 538.962,A -85,B 0,C 180,E1 -12690,E2 -12690} C_VEL
LIN {X 0,Y 368.186,Z 538.589,A -85,B 0,C 180,E1 -12691.093,E2 -12691.093} C_VEL
LIN {X 0,Y 368.164,Z 537.79,A -85,B 0,C 180,E1 -12692.187,E2 -12692.187} C_VEL
LIN {X 0,Y 368.221,Z 536.557,A -85,B 0,C 180,E1 -12693.282,E2 -12693.282} C_VEL
LIN {X 0,Y 368.027,Z 533.874,A -85,B 0,C 180,E1 -12694.929,E2 -12694.929} C_VEL
LIN {X 0,Y 367.925,Z 529.983,A -85,B 0,C 180,E1 -12696.64,E2 -12696.64} C_VEL
LIN {X 0,Y 367.903,Z 525.259,A -85,B 0,C 180,E1 -12698.237,E2 -12698.237} C_VEL
LIN {X 0,Y 368.106,Z 517.938,A -85,B 0,C 180,E1 -12700.171,E2 -12700.171} C_VEL
LIN {X 0,Y 368.556,Z 509.981,A -85,B 0,C 180,E1 -12701.828,E2 -12701.828} C_VEL
LIN {X 0,Y 369.286,Z 500.551,A -85,B 0,C 180,E1 -12703.403,E2 -12703.403} C_VEL
LIN {X 0,Y 370.037,Z 490.878,A -85,B 0,C 180,E1 -12704.715,E2 -12704.715} C_VEL
LIN {X 0,Y 370.985,Z 479.578,A -85,B 0,C 180,E1 -12705.943,E2 -12705.943} C_VEL
LIN {X 0,Y 371.937,Z 468.529,A -85,B 0,C 180,E1 -12706.888,E2 -12706.888} C_VEL
LIN {X 0,Y 372.924,Z 456.343,A -85,B 0,C 180,E1 -12707.69,E2 -12707.69} C_VEL
LIN {X 0,Y 373.687,Z 443.78,A -85,B 0,C 180,E1 -12708.29,E2 -12708.29} C_VEL
LIN {X 0,Y 374.095,Z 431.002,A -85,B 0,C 180,E1 -12708.686,E2 -12708.686} C_VEL
LIN {X 0,Y 374.822,Z 367.007,A -85,B 0,C 180,E1 -12709.914,E2 -12709.914} C_VEL
LIN {X 0,Y 370.295,Z 323.034,A -85,B 0,C 180,E1 -12711.017,E2 -12711.017} C_VEL
LIN {X 0,Y 371.787,Z 299.847,A -85,B 0,C 180,E1 -12714.955,E2 -12714.955} C_VEL
LIN {X 0,Y 373.066,Z 281.608,A -85,B 0,C 180,E1 -12718.096,E2 -12718.096} C_VEL
LIN {X 0,Y 372.807,Z 278.095,A -85,B 0,C 180,E1 -12718.731,E2 -12718.731} C_VEL
LIN {X 0,Y 369.656,Z 262.86,A -85,B 0,C 180,E1 -12721.646,E2 -12721.646} C_VEL
LIN {X 0,Y 368.931,Z 259.631,A -85,B 0,C 180,E1 -12722.335,E2 -12722.335} C_VEL
LIN {X 0,Y 368.918,Z 259.532,A -85,B 0,C 180,E1 -12724.999,E2 -12724.999} C_VEL
LIN {X 0,Y 368.868,Z 259.534,A -85,B 0,C 180,E1 -12728.632,E2 -12728.632} C_VEL
LIN {X 0,Y 368.851,Z 259.536,A -85,B 0,C 180,E1 -12732.004,E2 -12732.004} C_VEL
LIN {X 0,Y 368.866,Z 259.54,A -85,B 0,C 180,E1 -12735.174,E2 -12735.174} C_VEL
LIN {X 0,Y 368.852,Z 259.536,A -85,B 0,C 180,E1 -12738.173,E2 -12738.173} C_VEL
LIN {X 0,Y 368.867,Z 259.538,A -85,B 0,C 180,E1 -12741.365,E2 -12741.365} C_VEL
LIN {X 0,Y 368.921,Z 259.533,A -85,B 0,C 180,E1 -12745.145,E2 -12745.145} C_VEL
LIN {X 0,Y 368.886,Z 259.538,A -85,B 0,C 180,E1 -12749.043,E2 -12749.043} C_VEL
LIN {X 0,Y 368.896,Z 259.531,A -85,B 0,C 180,E1 -12751.557,E2 -12751.557} C_VEL
LIN {X 0,Y 368.911,Z 259.531,A -85,B 0,C 180,E1 -12755.221,E2 -12755.221} C_VEL
LIN {X 0,Y 368.909,Z 259.534,A -85,B 0,C 180,E1 -12758.98,E2 -12758.98} C_VEL
LIN {X 0,Y 368.98,Z 259.521,A -85,B 0,C 180,E1 -12762.257,E2 -12762.257} C_VEL
LIN {X 0,Y 369.026,Z 259.515,A -85,B 0,C 180,E1 -12766.228,E2 -12766.228} C_VEL
LIN {X 0,Y 369.048,Z 259.513,A -85,B 0,C 180,E1 -12770.131,E2 -12770.131} C_VEL
LIN {X 0,Y 369.139,Z 259.5,A -85,B 0,C 180,E1 -12773.441,E2 -12773.441} C_VEL
LIN {X 0,Y 369.292,Z 259.481,A -85,B 0,C 180,E1 -12777.819,E2 -12777.819} C_VEL
LIN {X 0,Y 369.282,Z 259.485,A -85,B 0,C 180,E1 -12782.182,E2 -12782.182} C_VEL
LIN {X 0,Y 369.141,Z 259.504,A -85,B 0,C 180,E1 -12786.568,E2 -12786.568} C_VEL
LIN {X 0,Y 369.045,Z 259.513,A -85,B 0,C 180,E1 -12789.869,E2 -12789.869} C_VEL
LIN {X 0,Y 369.027,Z 259.515,A -85,B 0,C 180,E1 -12793.772,E2 -12793.772} C_VEL
LIN {X 0,Y 368.981,Z 259.521,A -85,B 0,C 180,E1 -12797.744,E2 -12797.744} C_VEL
LIN {X 0,Y 368.9,Z 259.53,A -85,B 0,C 180,E1 -12801.222,E2 -12801.222} C_VEL
LIN {X 0,Y 368.907,Z 259.533,A -85,B 0,C 180,E1 -12803.877,E2 -12803.877} C_VEL
LIN {X 0,Y 368.848,Z 259.536,A -85,B 0,C 180,E1 -12807.213,E2 -12807.213} C_VEL
LIN {X 0,Y 368.884,Z 259.535,A -85,B 0,C 180,E1 -12809.694,E2 -12809.694} C_VEL
LIN {X 0,Y 368.888,Z 259.531,A -85,B 0,C 180,E1 -12813.044,E2 -12813.044} C_VEL
LIN {X 0,Y 368.903,Z 259.533,A -85,B 0,C 180,E1 -12816.199,E2 -12816.199} C_VEL
LIN {X 0,Y 368.866,Z 259.534,A -85,B 0,C 180,E1 -12818.958,E2 -12818.958} C_VEL
LIN {X 0,Y 368.852,Z 259.54,A -85,B 0,C 180,E1 -12822.006,E2 -12822.006} C_VEL
LIN {X 0,Y 368.867,Z 259.535,A -85,B 0,C 180,E1 -12825.176,E2 -12825.176} C_VEL
LIN {X 0,Y 368.855,Z 259.537,A -85,B 0,C 180,E1 -12828.176,E2 -12828.176} C_VEL
LIN {X 0,Y 368.872,Z 259.536,A -85,B 0,C 180,E1 -12831.368,E2 -12831.368} C_VEL
LIN {X 0,Y 368.928,Z 259.528,A -85,B 0,C 180,E1 -12835.147,E2 -12835.147} C_VEL
LIN {X 0,Y 368.894,Z 259.532,A -85,B 0,C 180,E1 -12839.045,E2 -12839.045} C_VEL
LIN {X 0,Y 368.905,Z 259.535,A -85,B 0,C 180,E1 -12841.559,E2 -12841.559} C_VEL
LIN {X 0,Y 368.884,Z 259.536,A -85,B 0,C 180,E1 -12845.22,E2 -12845.22} C_VEL
LIN {X 0,Y 368.916,Z 259.532,A -85,B 0,C 180,E1 -12847.605,E2 -12847.605} C_VEL
LIN {X 0,Y 368.907,Z 259.533,A -85,B 0,C 180,E1 -12851.104,E2 -12851.104} C_VEL
LIN {X 0,Y 368.928,Z 259.526,A -85,B 0,C 180,E1 -12854.533,E2 -12854.533} C_VEL
LIN {X 0,Y 369.055,Z 259.663,A -85,B 0,C 180,E1 -12857.281,E2 -12857.281} C_VEL
LIN {X 0,Y 369.304,Z 260.788,A -85,B 0,C 180,E1 -12857.477,E2 -12857.477} C_VEL
LIN {X 0,Y 376,Z 278.908,A -85,B 0,C 180,E1 -12858.189,E2 -12858.189} C_VEL
LIN {X 0,Y 375.048,Z 347.052,A -85,B 0,C 180,E1 -12859.508,E2 -12859.508} C_VEL
LIN {X 0,Y 374.868,Z 360.169,A -85,B 0,C 180,E1 -12859.98,E2 -12859.98} C_VEL
LIN {X 0,Y 374.526,Z 371.099,A -85,B 0,C 180,E1 -12860.55,E2 -12860.55} C_VEL
LIN {X 0,Y 373.974,Z 382.7,A -85,B 0,C 180,E1 -12861.354,E2 -12861.354} C_VEL
LIN {X 0,Y 373.306,Z 393.272,A -85,B 0,C 180,E1 -12862.292,E2 -12862.292} C_VEL
LIN {X 0,Y 372.509,Z 404.071,A -85,B 0,C 180,E1 -12863.501,E2 -12863.501} C_VEL
LIN {X 0,Y 371.776,Z 413.714,A -85,B 0,C 180,E1 -12864.849,E2 -12864.849} C_VEL
LIN {X 0,Y 370.963,Z 423.076,A -85,B 0,C 180,E1 -12866.47,E2 -12866.47} C_VEL
LIN {X 0,Y 370.171,Z 430.549,A -85,B 0,C 180,E1 -12868.096,E2 -12868.096} C_VEL
LIN {X 0,Y 369.686,Z 435.663,A -85,B 0,C 180,E1 -12869.456,E2 -12869.456} C_VEL
LIN {X 0,Y 369.232,Z 440.619,A -85,B 0,C 180,E1 -12871.091,E2 -12871.091} C_VEL
LIN {X 0,Y 368.884,Z 444.474,A -85,B 0,C 180,E1 -12872.73,E2 -12872.73} C_VEL
LIN {X 0,Y 368.7,Z 447.318,A -85,B 0,C 180,E1 -12874.373,E2 -12874.373} C_VEL
LIN {X 0,Y 368.678,Z 448.66,A -85,B 0,C 180,E1 -12875.47,E2 -12875.47} C_VEL
LIN {X 0,Y 368.618,Z 450.221,A -85,B 0,C 180,E1 -12877.67,E2 -12877.67} C_VEL
LIN {X 0,Y 368.639,Z 450.406,A -85,B 0,C 180,E1 -12878.773,E2 -12878.773} C_VEL
